LIN {X 0,Y 306.551,Z 155.301,A -85,B 0,C 180,E1 -15794.918,E2 -15794.918} C_VEL
LIN {X 0,Y 305.506,Z 155.43,A -85,B 0,C 180,E1 -15796.018,E2 -15796.018} C_VEL
LIN {X 0,Y 305.419,Z 155.438,A -85,B 0,C 180,E1 -15796.391,E2 -15796.391} C_VEL
LIN {X 0,Y 305.452,Z 155.438,A -85,B 0,C 180,E1 -15799.891,E2 -15799.891} C_VEL
LIN {X 0,Y 305.474,Z 155.435,A -85,B 0,C 180,E1 -15803.63,E2 -15803.63} C_VEL
LIN {X 0,Y 305.457,Z 155.432,A -85,B 0,C 180,E1 -15806.482,E2 -15806.482} C_VEL
LIN {X 0,Y 305.455,Z 155.439,A -85,B 0,C 180,E1 -15809.59,E2 -15809.59} C_VEL
LIN {X 0,Y 305.482,Z 155.427,A -85,B 0,C 180,E1 -15812.604,E2 -15812.604} C_VEL
LIN {X 0,Y 305.483,Z 155.435,A -85,B 0,C 180,E1 -15815.536,E2 -15815.536} C_VEL
LIN {X 0,Y 305.475,Z 155.433,A -85,B 0,C 180,E1 -15819.812,E2 -15819.812} C_VEL
LIN {X 0,Y 305.54,Z 155.42,A -85,B 0,C 180,E1 -15823.977,E2 -15823.977} C_VEL
LIN {X 0,Y 305.576,Z 155.419,A -85,B 0,C 180,E1 -15826.703,E2 -15826.703} C_VEL
LIN {X 0,Y 305.742,Z 155.395,A -85,B 0,C 180,E1 -15831.261,E2 -15831.261} C_VEL
LIN {X 0,Y 305.773,Z 155.383,A -85,B 0,C 180,E1 -15833.401,E2 -15833.401} C_VEL
LIN {X 0,Y 305.923,Z 155.375,A -85,B 0,C 180,E1 -15838.683,E2 -15838.683} C_VEL
LIN {X 0,Y 305.923,Z 155.377,A -85,B 0,C 180,E1 -15841.316,E2 -15841.316} C_VEL
LIN {X 0,Y 305.775,Z 155.396,A -85,B 0,C 180,E1 -15846.599,E2 -15846.599} C_VEL
LIN {X 0,Y 305.684,Z 155.408,A -85,B 0,C 180,E1 -15849.261,E2 -15849.261} C_VEL
LIN {X 0,Y 305.576,Z 155.421,A -85,B 0,C 180,E1 -15853.297,E2 -15853.297} C_VEL
LIN {X 0,Y 305.54,Z 155.423,A -85,B 0,C 180,E1 -15856.023,E2 -15856.023} C_VEL
LIN {X 0,Y 305.474,Z 155.433,A -85,B 0,C 180,E1 -15860.188,E2 -15860.188} C_VEL
LIN {X 0,Y 305.482,Z 155.435,A -85,B 0,C 180,E1 -15864.463,E2 -15864.463} C_VEL
LIN {X 0,Y 305.481,Z 155.432,A -85,B 0,C 180,E1 -15867.395,E2 -15867.395} C_VEL
LIN {X 0,Y 305.454,Z 155.44,A -85,B 0,C 180,E1 -15870.41,E2 -15870.41} C_VEL
LIN {X 0,Y 305.456,Z 155.437,A -85,B 0,C 180,E1 -15874.079,E2 -15874.079} C_VEL
LIN {X 0,Y 305.467,Z 155.436,A -85,B 0,C 180,E1 -15876.741,E2 -15876.741} C_VEL
LIN {X 0,Y 305.447,Z 155.438,A -85,B 0,C 180,E1 -15880.601,E2 -15880.601} C_VEL
LIN {X 0,Y 305.419,Z 155.44,A -85,B 0,C 180,E1 -15883.656,E2 -15883.656} C_VEL
LIN {X 0,Y 305.449,Z 155.434,A -85,B 0,C 180,E1 -15887.416,E2 -15887.416} C_VEL
LIN {X 0,Y 305.49,Z 155.431,A -85,B 0,C 180,E1 -15891.602,E2 -15891.602} C_VEL
LIN {X 0,Y 305.458,Z 155.437,A -85,B 0,C 180,E1 -15894.888,E2 -15894.888} C_VEL
LIN {X 0,Y 305.514,Z 155.509,A -85,B 0,C 180,E1 -15897.229,E2 -15897.229} C_VEL
LIN {X 0,Y 308.104,Z 167.27,A -85,B 0,C 180,E1 -15900.722,E2 -15900.722} C_VEL
LIN {X 0,Y 309.757,Z 176.68,A -85,B 0,C 180,E1 -15903.38,E2 -15903.38} C_VEL
LIN {X 0,Y 309.124,Z 182.65,A -85,B 0,C 180,E1 -15904.915,E2 -15904.915} C_VEL
LIN {X 0,Y 313.255,Z 210.257,A -85,B 0,C 180,E1 -15905.903,E2 -15905.903} C_VEL
LIN {X 0,Y 315.301,Z 227.992,A -85,B 0,C 180,E1 -15906.476,E2 -15906.476} C_VEL
LIN {X 0,Y 313.856,Z 291.58,A -85,B 0,C 180,E1 -15907.93,E2 -15907.93} C_VEL
LIN {X 0,Y 313.125,Z 304.866,A -85,B 0,C 180,E1 -15908.481,E2 -15908.481} C_VEL
LIN {X 0,Y 312.062,Z 317.037,A -85,B 0,C 180,E1 -15909.226,E2 -15909.226} C_VEL
LIN {X 0,Y 310.871,Z 328.51,A -85,B 0,C 180,E1 -15910.179,E2 -15910.179} C_VEL
LIN {X 0,Y 309.461,Z 340.297,A -85,B 0,C 180,E1 -15911.463,E2 -15911.463} C_VEL
LIN {X 0,Y 308.023,Z 350.876,A -85,B 0,C 180,E1 -15912.918,E2 -15912.918} C_VEL
LIN {X 0,Y 307.034,Z 359.54,A -85,B 0,C 180,E1 -15914.399,E2 -15914.399} C_VEL
LIN {X 0,Y 305.962,Z 367.513,A -85,B 0,C 180,E1 -15916.045,E2 -15916.045} C_VEL
LIN {X 0,Y 304.92,Z 375.297,A -85,B 0,C 180,E1 -15918.029,E2 -15918.029} C_VEL
LIN {X 0,Y 304.28,Z 381.547,A -85,B 0,C 180,E1 -15920.026,E2 -15920.026} C_VEL
LIN {X 0,Y 303.88,Z 386.51,A -85,B 0,C 180,E1 -15922.025,E2 -15922.025} C_VEL
LIN {X 0,Y 303.73,Z 390.71,A -85,B 0,C 180,E1 -15924.256,E2 -15924.256} C_VEL
LIN {X 0,Y 303.707,Z 393.121,A -85,B 0,C 180,E1 -15926.02,E2 -15926.02} C_VEL
LIN {X 0,Y 303.689,Z 394.432,A -85,B 0,C 180,E1 -15927.348,E2 -15927.348} C_VEL
LIN {X 0,Y 303.699,Z 395.344,A -85,B 0,C 180,E1 -15928.675,E2 -15928.675} C_VEL
LIN {X 0,Y 303.761,Z 395.844,A -85,B 0,C 180,E1 -15930.001,E2 -15930.001} C_VEL
LIN {X 0,Y 303.684,Z 395.908,A -85,B 0,C 180,E1 -15931.327,E2 -15931.327} C_VEL
LIN {X 0,Y 303.656,Z 395.586,A -85,B 0,C 180,E1 -15932.654,E2 -15932.654} C_VEL
LIN {X 0,Y 303.651,Z 394.878,A -85,B 0,C 180,E1 -15933.983,E2 -15933.983} C_VEL
LIN {X 0,Y 303.619,Z 393.522,A -85,B 0,C 180,E1 -15935.533,E2 -15935.533} C_VEL
LIN {X 0,Y 303.915,Z 390.231,A -85,B 0,C 180,E1 -15937.977,E2 -15937.977} C_VEL
LIN {X 0,Y 304.375,Z 386.422,A -85,B 0,C 180,E1 -15939.974,E2 -15939.974} C_VEL
LIN {X 0,Y 305.103,Z 381.502,A -85,B 0,C 180,E1 -15941.966,E2 -15941.966} C_VEL
LIN {X 0,Y 306.325,Z 375.332,A -85,B 0,C 180,E1 -15943.941,E2 -15943.941} C_VEL
LIN {X 0,Y 307.732,Z 367.675,A -85,B 0,C 180,E1 -15945.907,E2 -15945.907} C_VEL
LIN {X 0,Y 309.092,Z 359.858,A -85,B 0,C 180,E1 -15947.535,E2 -15947.535} C_VEL
LIN {X 0,Y 310.844,Z 350.334,A -85,B 0,C 180,E1 -15949.138,E2 -15949.138} C_VEL
LIN {X 0,Y 312.706,Z 339.792,A -85,B 0,C 180,E1 -15950.56,E2 -15950.56} C_VEL
LIN {X 0,Y 314.494,Z 328.047,A -85,B 0,C 180,E1 -15951.81,E2 -15951.81} C_VEL
LIN {X 0,Y 316.168,Z 315.476,A -85,B 0,C 180,E1 -15952.807,E2 -15952.807} C_VEL
LIN {X 0,Y 317.508,Z 302.295,A -85,B 0,C 180,E1 -15953.562,E2 -15953.562} C_VEL
LIN {X 0,Y 318.318,Z 289.851,A -85,B 0,C 180,E1 -15954.027,E2 -15954.027} C_VEL
LIN {X 0,Y 319.87,Z 227.886,A -85,B 0,C 180,E1 -15955.437,E2 -15955.437} C_VEL
LIN {X 0,Y 316.156,Z 205.273,A -85,B 0,C 180,E1 -15956.354,E2 -15956.354} C_VEL
LIN {X 0,Y 311.988,Z 184.189,A -85,B 0,C 180,E1 -15957.307,E2 -15957.307} C_VEL
LIN {X 0,Y 311.433,Z 182.073,A -85,B 0,C 180,E1 -15957.456,E2 -15957.456} C_VEL
LIN {X 0,Y 309.514,Z 172.334,A -85,B 0,C 180,E1 -15960.362,E2 -15960.362} C_VEL
LIN {X 0,Y 307.088,Z 161.825,A -85,B 0,C 180,E1 -15963.682,E2 -15963.682} C_VEL
LIN {X 0,Y 305.495,Z 155.433,A -85,B 0,C 180,E1 -15965.818,E2 -15965.818} C_VEL
LIN {X 0,Y 305.469,Z 155.43,A -85,B 0,C 180,E1 -15968.533,E2 -15968.533} C_VEL
LIN {X 0,Y 305.457,Z 155.433,A -85,B 0,C 180,E1 -15972.586,E2 -15972.586} C_VEL
LIN {X 0,Y 305.424,Z 155.44,A -85,B 0,C 180,E1 -15976.345,E2 -15976.345} C_VEL
LIN {X 0,Y 305.412,Z 155.443,A -85,B 0,C 180,E1 -15979.885,E2 -15979.885} C_VEL
LIN {X 0,Y 305.464,Z 155.437,A -85,B 0,C 180,E1 -15983.637,E2 -15983.637} C_VEL
LIN {X 0,Y 305.467,Z 155.436,A -85,B 0,C 180,E1 -15986.483,E2 -15986.483} C_VEL
LIN {X 0,Y 305.432,Z 155.439,A -85,B 0,C 180,E1 -15989.588,E2 -15989.588} C_VEL
LIN {X 0,Y 305.458,Z 155.436,A -85,B 0,C 180,E1 -15992.603,E2 -15992.603} C_VEL
LIN {X 0,Y 305.475,Z 155.432,A -85,B 0,C 180,E1 -15995.536,E2 -15995.536} C_VEL
LIN {X 0,Y 305.461,Z 155.436,A -85,B 0,C 180,E1 -15998.4,E2 -15998.4} C_VEL
LIN {X 0,Y 305.51,Z 155.421,A -85,B 0,C 180,E1 -16001.213,E2 -16001.213} C_VEL
LIN {X 0,Y 305.571,Z 155.41,A -85,B 0,C 180,E1 -16005.345,E2 -16005.345} C_VEL
LIN {X 0,Y 305.623,Z 155.413,A -85,B 0,C 180,E1 -16009.399,E2 -16009.399} C_VEL
LIN {X 0,Y 305.739,Z 155.389,A -85,B 0,C 180,E1 -16012.073,E2 -16012.073} C_VEL
LIN {X 0,Y 305.654,Z 155.41,A -85,B 0,C 180,E1 -16014.723,E2 -16014.723} C_VEL
LIN {X 0,Y 305.932,Z 155.374,A -85,B 0,C 180,E1 -16018.684,E2 -16018.684} C_VEL
LIN {X 0,Y 305.935,Z 155.375,A -85,B 0,C 180,E1 -16021.316,E2 -16021.316} C_VEL
LIN {X 0,Y 305.787,Z 155.392,A -85,B 0,C 180,E1 -16026.599,E2 -16026.599} C_VEL
LIN {X 0,Y 305.696,Z 155.394,A -85,B 0,C 180,E1 -16029.261,E2 -16029.261} C_VEL
LIN {X 0,Y 305.587,Z 155.412,A -85,B 0,C 180,E1 -16033.296,E2 -16033.296} C_VEL
LIN {X 0,Y 305.553,Z 155.423,A -85,B 0,C 180,E1 -16036.022,E2 -16036.022} C_VEL
LIN {X 0,Y 305.486,Z 155.425,A -85,B 0,C 180,E1 -16040.188,E2 -16040.188} C_VEL
LIN {X 0,Y 305.489,Z 155.429,A -85,B 0,C 180,E1 -16043.039,E2 -16043.039} C_VEL
LIN {X 0,Y 305.476,Z 155.432,A -85,B 0,C 180,E1 -16046.198,E2 -16046.198} C_VEL
LIN {X 0,Y 305.465,Z 155.429,A -85,B 0,C 180,E1 -16049.038,E2 -16049.038} C_VEL
LIN {X 0,Y 305.44,Z 155.435,A -85,B 0,C 180,E1 -16051.953,E2 -16051.953} C_VEL
LIN {X 0,Y 305.465,Z 155.433,A -85,B 0,C 180,E1 -16055.113,E2 -16055.113} C_VEL
LIN {X 0,Y 305.453,Z 155.436,A -85,B 0,C 180,E1 -16058.529,E2 -16058.529} C_VEL
LIN {X 0,Y 305.458,Z 155.424,A -85,B 0,C 180,E1 -16062.586,E2 -16062.586} C_VEL
LIN {X 0,Y 305.429,Z 155.442,A -85,B 0,C 180,E1 -16066.345,E2 -16066.345} C_VEL
LIN {X 0,Y 305.462,Z 155.435,A -85,B 0,C 180,E1 -16069.892,E2 -16069.892} C_VEL
LIN {X 0,Y 305.484,Z 155.434,A -85,B 0,C 180,E1 -16073.632,E2 -16073.632} C_VEL
LIN {X 0,Y 305.481,Z 155.444,A -85,B 0,C 180,E1 -16076.12,E2 -16076.12} C_VEL
LIN {X 0,Y 306.181,Z 158.233,A -85,B 0,C 180,E1 -16077.073,E2 -16077.073} C_VEL
LIN {X 0,Y 315.619,Z 178.208,A -85,B 0,C 180,E1 -16078.583,E2 -16078.583} C_VEL
LIN {X 0,Y 320.869,Z 190.79,A -85,B 0,C 180,E1 -16079.412,E2 -16079.412} C_VEL
LIN {X 0,Y 318.922,Z 264.646,A -85,B 0,C 180,E1 -16081.089,E2 -16081.089} C_VEL
LIN {X 0,Y 318.114,Z 278.09,A -85,B 0,C 180,E1 -16081.64,E2 -16081.64} C_VEL
LIN {X 0,Y 316.947,Z 290.836,A -85,B 0,C 180,E1 -16082.42,E2 -16082.42} C_VEL
LIN {X 0,Y 315.814,Z 301.857,A -85,B 0,C 180,E1 -16083.35,E2 -16083.35} C_VEL
LIN {X 0,Y 314.305,Z 312.622,A -85,B 0,C 180,E1 -16084.504,E2 -16084.504} C_VEL
LIN {X 0,Y 312.461,Z 323.31,A -85,B 0,C 180,E1 -16085.94,E2 -16085.94} C_VEL
LIN {X 0,Y 310.788,Z 333.59,A -85,B 0,C 180,E1 -16087.703,E2 -16087.703} C_VEL
LIN {X 0,Y 309.416,Z 341.439,A -85,B 0,C 180,E1 -16089.385,E2 -16089.385} C_VEL
LIN {X 0,Y 307.799,Z 348.931,A -85,B 0,C 180,E1 -16091.356,E2 -16091.356} C_VEL
LIN {X 0,Y 306.52,Z 354.927,A -85,B 0,C 180,E1 -16093.344,E2 -16093.344} C_VEL
LIN {X 0,Y 305.543,Z 359.651,A -85,B 0,C 180,E1 -16095.343,E2 -16095.343} C_VEL
LIN {X 0,Y 304.823,Z 363.251,A -85,B 0,C 180,E1 -16097.347,E2 -16097.347} C_VEL
LIN {X 0,Y 304.261,Z 365.832,A -85,B 0,C 180,E1 -16099.35,E2 -16099.35} C_VEL
LIN {X 0,Y 304.05,Z 367.039,A -85,B 0,C 180,E1 -16100.687,E2 -16100.687} C_VEL
LIN {X 0,Y 303.936,Z 367.823,A -85,B 0,C 180,E1 -16102.024,E2 -16102.024} C_VEL
LIN {X 0,Y 303.915,Z 368.252,A -85,B 0,C 180,E1 -16103.921,E2 -16103.921} C_VEL
LIN {X 0,Y 303.824,Z 367.797,A -85,B 0,C 180,E1 -16106.02,E2 -16106.02} C_VEL
LIN {X 0,Y 303.764,Z 367.012,A -85,B 0,C 180,E1 -16107.347,E2 -16107.347} C_VEL
LIN {X 0,Y 303.999,Z 364.191,A -85,B 0,C 180,E1 -16109.999,E2 -16109.999} C_VEL
LIN {X 0,Y 304.334,Z 360.97,A -85,B 0,C 180,E1 -16111.984,E2 -16111.984} C_VEL
LIN {X 0,Y 304.854,Z 356.695,A -85,B 0,C 180,E1 -16113.965,E2 -16113.965} C_VEL
LIN {X 0,Y 305.747,Z 350.237,A -85,B 0,C 180,E1 -16116.267,E2 -16116.267} C_VEL
LIN {X 0,Y 306.744,Z 343.147,A -85,B 0,C 180,E1 -16118.232,E2 -16118.232} C_VEL
LIN {X 0,Y 307.877,Z 335.937,A -85,B 0,C 180,E1 -16119.857,E2 -16119.857} C_VEL
LIN {X 0,Y 308.713,Z 329.148,A -85,B 0,C 180,E1 -16121.156,E2 -16121.156} C_VEL
LIN {X 0,Y 310.118,Z 318.516,A -85,B 0,C 180,E1 -16122.807,E2 -16122.807} C_VEL
LIN {X 0,Y 311.431,Z 307.191,A -85,B 0,C 180,E1 -16124.205,E2 -16124.205} C_VEL
LIN {X 0,Y 312.562,Z 295.58,A -85,B 0,C 180,E1 -16125.318,E2 -16125.318} C_VEL
LIN {X 0,Y 313.407,Z 283.539,A -85,B 0,C 180,E1 -16126.193,E2 -16126.193} C_VEL
LIN {X 0,Y 314.141,Z 270.385,A -85,B 0,C 180,E1 -16126.865,E2 -16126.865} C_VEL
LIN {X 0,Y 314.557,Z 256.796,A -85,B 0,C 180,E1 -16127.277,E2 -16127.277} C_VEL
LIN {X 0,Y 316.158,Z 186.608,A -85,B 0,C 180,E1 -16128.846,E2 -16128.846} C_VEL
LIN {X 0,Y 314.888,Z 180.875,A -85,B 0,C 180,E1 -16129.078,E2 -16129.078} C_VEL
LIN {X 0,Y 307.233,Z 160.574,A -85,B 0,C 180,E1 -16130.17,E2 -16130.17} C_VEL
LIN {X 0,Y 305.968,Z 157.454,A -85,B 0,C 180,E1 -16130.371,E2 -16130.371} C_VEL
LIN {X 0,Y 305.517,Z 155.429,A -85,B 0,C 180,E1 -16131.063,E2 -16131.063} C_VEL
LIN {X 0,Y 305.504,Z 155.432,A -85,B 0,C 180,E1 -16134.46,E2 -16134.46} C_VEL
LIN {X 0,Y 305.52,Z 155.426,A -85,B 0,C 180,E1 -16137.39,E2 -16137.39} C_VEL
LIN {X 0,Y 305.461,Z 155.436,A -85,B 0,C 180,E1 -16140.407,E2 -16140.407} C_VEL
LIN {X 0,Y 305.461,Z 155.436,A -85,B 0,C 180,E1 -16144.077,E2 -16144.077} C_VEL
LIN {X 0,Y 305.476,Z 155.431,A -85,B 0,C 180,E1 -16146.737,E2 -16146.737} C_VEL
LIN {X 0,Y 305.45,Z 155.434,A -85,B 0,C 180,E1 -16150.598,E2 -16150.598} C_VEL
LIN {X 0,Y 305.42,Z 155.441,A -85,B 0,C 180,E1 -16153.654,E2 -16153.654} C_VEL
LIN {X 0,Y 305.419,Z 155.438,A -85,B 0,C 180,E1 -16156.391,E2 -16156.391} C_VEL
LIN {X 0,Y 304.737,Z 155.524,A -85,B 0,C 180,E1 -16157.491,E2 -16157.491} C_VEL
LIN {X 0,Y 301.866,Z 155.882,A -85,B 0,C 180,E1 -16159.282,E2 -16159.282} C_VEL
LIN {X 0,Y 299.466,Z 156.179,A -85,B 0,C 180,E1 -16160.735,E2 -16160.735} C_VEL
LIN {X 0,Y 298.477,Z 156.305,A -85,B 0,C 180,E1 -16161.86,E2 -16161.86} C_VEL
LIN {X 0,Y 298.418,Z 156.311,A -85,B 0,C 180,E1 -16162.241,E2 -16162.241} C_VEL
LIN {X 0,Y 298.401,Z 156.317,A -85,B 0,C 180,E1 -16165.58,E2 -16165.58} C_VEL
LIN {X 0,Y 298.387,Z 156.314,A -85,B 0,C 180,E1 -16168.79,E2 -16168.79} C_VEL
LIN {X 0,Y 298.439,Z 156.307,A -85,B 0,C 180,E1 -16171.902,E2 -16171.902} C_VEL
LIN {X 0,Y 298.457,Z 156.306,A -85,B 0,C 180,E1 -16174.921,E2 -16174.921} C_VEL
LIN {X 0,Y 298.413,Z 156.311,A -85,B 0,C 180,E1 -16179.312,E2 -16179.312} C_VEL
LIN {X 0,Y 298.456,Z 156.305,A -85,B 0,C 180,E1 -16182.174,E2 -16182.174} C_VEL
LIN {X 0,Y 298.576,Z 156.289,A -85,B 0,C 180,E1 -16184.994,E2 -16184.994} C_VEL
LIN {X 0,Y 298.573,Z 156.295,A -85,B 0,C 180,E1 -16189.146,E2 -16189.146} C_VEL
LIN {X 0,Y 298.686,Z 156.268,A -85,B 0,C 180,E1 -16191.884,E2 -16191.884} C_VEL
LIN {X 0,Y 298.615,Z 156.271,A -85,B 0,C 180,E1 -16194.598,E2 -16194.598} C_VEL
LIN {X 0,Y 298.891,Z 156.251,A -85,B 0,C 180,E1 -16198.652,E2 -16198.652} C_VEL
LIN {X 0,Y 298.891,Z 156.253,A -85,B 0,C 180,E1 -16201.347,E2 -16201.347} C_VEL
LIN {X 0,Y 298.724,Z 156.276,A -85,B 0,C 180,E1 -16206.755,E2 -16206.755} C_VEL
LIN {X 0,Y 298.615,Z 156.287,A -85,B 0,C 180,E1 -16209.482,E2 -16209.482} C_VEL
LIN {X 0,Y 298.535,Z 156.297,A -85,B 0,C 180,E1 -16213.616,E2 -16213.616} C_VEL
LIN {X 0,Y 298.474,Z 156.306,A -85,B 0,C 180,E1 -16216.413,E2 -16216.413} C_VEL
LIN {X 0,Y 298.45,Z 156.307,A -85,B 0,C 180,E1 -16219.627,E2 -16219.627} C_VEL
LIN {X 0,Y 298.416,Z 156.312,A -85,B 0,C 180,E1 -16223.601,E2 -16223.601} C_VEL
LIN {X 0,Y 298.447,Z 156.313,A -85,B 0,C 180,E1 -16226.578,E2 -16226.578} C_VEL
LIN {X 0,Y 298.411,Z 156.313,A -85,B 0,C 180,E1 -16229.642,E2 -16229.642} C_VEL
LIN {X 0,Y 298.387,Z 156.318,A -85,B 0,C 180,E1 -16232.801,E2 -16232.801} C_VEL
LIN {X 0,Y 298.438,Z 156.311,A -85,B 0,C 180,E1 -16236.809,E2 -16236.809} C_VEL
LIN {X 0,Y 298.38,Z 156.316,A -85,B 0,C 180,E1 -16241.089,E2 -16241.089} C_VEL
LIN {X 0,Y 298.392,Z 156.314,A -85,B 0,C 180,E1 -16243.105,E2 -16243.105} C_VEL
LIN {X 0,Y 298.397,Z 156.312,A -85,B 0,C 180,E1 -16246.922,E2 -16246.922} C_VEL
LIN {X 0,Y 298.41,Z 156.312,A -85,B 0,C 180,E1 -16251.005,E2 -16251.005} C_VEL
LIN {X 0,Y 298.427,Z 156.314,A -85,B 0,C 180,E1 -16253.934,E2 -16253.934} C_VEL
LIN {X 0,Y 298.463,Z 156.476,A -85,B 0,C 180,E1 -16256.808,E2 -16256.808} C_VEL
LIN {X 0,Y 300.859,Z 167.223,A -85,B 0,C 180,E1 -16260.1,E2 -16260.1} C_VEL
LIN {X 0,Y 302.772,Z 177.488,A -85,B 0,C 180,E1 -16263.089,E2 -16263.089} C_VEL
LIN {X 0,Y 302.362,Z 182.254,A -85,B 0,C 180,E1 -16264.353,E2 -16264.353} C_VEL
LIN {X 0,Y 306.762,Z 211.709,A -85,B 0,C 180,E1 -16265.456,E2 -16265.456} C_VEL
LIN {X 0,Y 308.696,Z 228.156,A -85,B 0,C 180,E1 -16266.006,E2 -16266.006} C_VEL
LIN {X 0,Y 307.189,Z 291.052,A -85,B 0,C 180,E1 -16267.469,E2 -16267.469} C_VEL
LIN {X 0,Y 306.462,Z 304.412,A -85,B 0,C 180,E1 -16268.034,E2 -16268.034} C_VEL
LIN {X 0,Y 305.297,Z 317.183,A -85,B 0,C 180,E1 -16268.832,E2 -16268.832} C_VEL
LIN {X 0,Y 303.982,Z 329.327,A -85,B 0,C 180,E1 -16269.887,E2 -16269.887} C_VEL
LIN {X 0,Y 302.523,Z 340.894,A -85,B 0,C 180,E1 -16271.197,E2 -16271.197} C_VEL
LIN {X 0,Y 301.042,Z 351.528,A -85,B 0,C 180,E1 -16272.72,E2 -16272.72} C_VEL
LIN {X 0,Y 299.946,Z 360.695,A -85,B 0,C 180,E1 -16274.371,E2 -16274.371} C_VEL
LIN {X 0,Y 298.86,Z 368.395,A -85,B 0,C 180,E1 -16276.054,E2 -16276.054} C_VEL
LIN {X 0,Y 297.799,Z 375.939,A -85,B 0,C 180,E1 -16278.084,E2 -16278.084} C_VEL
LIN {X 0,Y 297.073,Z 382.914,A -85,B 0,C 180,E1 -16280.469,E2 -16280.469} C_VEL
LIN {X 0,Y 296.744,Z 387.511,A -85,B 0,C 180,E1 -16282.517,E2 -16282.517} C_VEL
LIN {X 0,Y 296.62,Z 391.004,A -85,B 0,C 180,E1 -16284.563,E2 -16284.563} C_VEL
LIN {X 0,Y 296.618,Z 392.745,A -85,B 0,C 180,E1 -16285.925,E2 -16285.925} C_VEL
LIN {X 0,Y 296.611,Z 394.068,A -85,B 0,C 180,E1 -16287.285,E2 -16287.285} C_VEL
LIN {X 0,Y 296.611,Z 394.992,A -85,B 0,C 180,E1 -16288.644,E2 -16288.644} C_VEL
LIN {X 0,Y 296.669,Z 395.513,A -85,B 0,C 180,E1 -16290.001,E2 -16290.001} C_VEL
LIN {X 0,Y 296.597,Z 395.591,A -85,B 0,C 180,E1 -16291.359,E2 -16291.359} C_VEL
LIN {X 0,Y 296.578,Z 395.28,A -85,B 0,C 180,E1 -16292.718,E2 -16292.718} C_VEL
LIN {X 0,Y 296.563,Z 394.582,A -85,B 0,C 180,E1 -16294.078,E2 -16294.078} C_VEL
LIN {X 0,Y 296.547,Z 393.419,A -85,B 0,C 180,E1 -16295.51,E2 -16295.51} C_VEL
LIN {X 0,Y 296.857,Z 389.983,A -85,B 0,C 180,E1 -16298.168,E2 -16298.168} C_VEL
LIN {X 0,Y 297.364,Z 386.2,A -85,B 0,C 180,E1 -16300.211,E2 -16300.211} C_VEL
LIN {X 0,Y 298.12,Z 381.308,A -85,B 0,C 180,E1 -16302.251,E2 -16302.251} C_VEL
LIN {X 0,Y 299.426,Z 375.169,A -85,B 0,C 180,E1 -16304.269,E2 -16304.269} C_VEL
LIN {X 0,Y 300.9,Z 367.555,A -85,B 0,C 180,E1 -16306.278,E2 -16306.278} C_VEL
LIN {X 0,Y 302.315,Z 359.785,A -85,B 0,C 180,E1 -16307.941,E2 -16307.941} C_VEL
LIN {X 0,Y 304.14,Z 350.323,A -85,B 0,C 180,E1 -16309.577,E2 -16309.577} C_VEL
LIN {X 0,Y 306.058,Z 339.845,A -85,B 0,C 180,E1 -16311.027,E2 -16311.027} C_VEL
LIN {X 0,Y 307.923,Z 328.207,A -85,B 0,C 180,E1 -16312.3,E2 -16312.3} C_VEL
LIN {X 0,Y 309.664,Z 315.813,A -85,B 0,C 180,E1 -16313.314,E2 -16313.314} C_VEL
LIN {X 0,Y 311.037,Z 302.848,A -85,B 0,C 180,E1 -16314.084,E2 -16314.084} C_VEL
LIN {X 0,Y 311.938,Z 289.634,A -85,B 0,C 180,E1 -16314.6,E2 -16314.6} C_VEL
LIN {X 0,Y 313.568,Z 228.936,A -85,B 0,C 180,E1 -16316.005,E2 -16316.005} C_VEL
LIN {X 0,Y 309.983,Z 206.806,A -85,B 0,C 180,E1 -16316.926,E2 -16316.926} C_VEL
LIN {X 0,Y 305.941,Z 186.404,A -85,B 0,C 180,E1 -16317.881,E2 -16317.881} C_VEL
LIN {X 0,Y 304.258,Z 181.669,A -85,B 0,C 180,E1 -16318.234,E2 -16318.234} C_VEL
LIN {X 0,Y 301.967,Z 170.913,A -85,B 0,C 180,E1 -16321.579,E2 -16321.579} C_VEL
LIN {X 0,Y 299.633,Z 161.081,A -85,B 0,C 180,E1 -16324.821,E2 -16324.821} C_VEL
LIN {X 0,Y 298.442,Z 156.306,A -85,B 0,C 180,E1 -16326.547,E2 -16326.547} C_VEL
LIN {X 0,Y 298.411,Z 156.307,A -85,B 0,C 180,E1 -16329.487,E2 -16329.487} C_VEL
LIN {X 0,Y 298.401,Z 156.314,A -85,B 0,C 180,E1 -16333.104,E2 -16333.104} C_VEL
LIN {X 0,Y 298.373,Z 156.32,A -85,B 0,C 180,E1 -16336.915,E2 -16336.915} C_VEL
LIN {X 0,Y 298.387,Z 156.317,A -85,B 0,C 180,E1 -16341.011,E2 -16341.011} C_VEL
LIN {X 0,Y 298.406,Z 156.315,A -85,B 0,C 180,E1 -16343.928,E2 -16343.928} C_VEL
LIN {X 0,Y 298.395,Z 156.316,A -85,B 0,C 180,E1 -16347.2,E2 -16347.2} C_VEL
LIN {X 0,Y 298.404,Z 156.316,A -85,B 0,C 180,E1 -16350.625,E2 -16350.625} C_VEL
LIN {X 0,Y 298.441,Z 156.311,A -85,B 0,C 180,E1 -16354.92,E2 -16354.92} C_VEL
LIN {X 0,Y 298.4,Z 156.314,A -85,B 0,C 180,E1 -16357.862,E2 -16357.862} C_VEL
LIN {X 0,Y 298.461,Z 156.296,A -85,B 0,C 180,E1 -16360.752,E2 -16360.752} C_VEL
LIN {X 0,Y 298.512,Z 156.291,A -85,B 0,C 180,E1 -16364.991,E2 -16364.991} C_VEL
LIN {X 0,Y 298.581,Z 156.291,A -85,B 0,C 180,E1 -16369.146,E2 -16369.146} C_VEL
LIN {X 0,Y 298.685,Z 156.267,A -85,B 0,C 180,E1 -16371.884,E2 -16371.884} C_VEL
LIN {X 0,Y 298.625,Z 156.286,A -85,B 0,C 180,E1 -16374.598,E2 -16374.598} C_VEL
LIN {X 0,Y 298.9,Z 156.25,A -85,B 0,C 180,E1 -16378.653,E2 -16378.653} C_VEL
LIN {X 0,Y 298.902,Z 156.251,A -85,B 0,C 180,E1 -16381.347,E2 -16381.347} C_VEL
LIN {X 0,Y 298.736,Z 156.271,A -85,B 0,C 180,E1 -16386.755,E2 -16386.755} C_VEL
LIN {X 0,Y 298.628,Z 156.276,A -85,B 0,C 180,E1 -16389.482,E2 -16389.482} C_VEL
LIN {X 0,Y 298.546,Z 156.286,A -85,B 0,C 180,E1 -16393.616,E2 -16393.616} C_VEL
LIN {X 0,Y 298.486,Z 156.303,A -85,B 0,C 180,E1 -16396.412,E2 -16396.412} C_VEL
LIN {X 0,Y 298.448,Z 156.299,A -85,B 0,C 180,E1 -16399.619,E2 -16399.619} C_VEL
LIN {X 0,Y 298.424,Z 156.304,A -85,B 0,C 180,E1 -16403.601,E2 -16403.601} C_VEL
LIN {X 0,Y 298.416,Z 156.313,A -85,B 0,C 180,E1 -16406.582,E2 -16406.582} C_VEL
LIN {X 0,Y 298.403,Z 156.312,A -85,B 0,C 180,E1 -16409.643,E2 -16409.643} C_VEL
LIN {X 0,Y 298.396,Z 156.31,A -85,B 0,C 180,E1 -16412.8,E2 -16412.8} C_VEL
LIN {X 0,Y 298.449,Z 156.304,A -85,B 0,C 180,E1 -16416.807,E2 -16416.807} C_VEL
LIN {X 0,Y 298.39,Z 156.293,A -85,B 0,C 180,E1 -16421.087,E2 -16421.087} C_VEL
LIN {X 0,Y 298.402,Z 156.311,A -85,B 0,C 180,E1 -16423.103,E2 -16423.103} C_VEL
LIN {X 0,Y 298.407,Z 156.313,A -85,B 0,C 180,E1 -16426.921,E2 -16426.921} C_VEL
LIN {X 0,Y 298.403,Z 156.314,A -85,B 0,C 180,E1 -16431.007,E2 -16431.007} C_VEL
LIN {X 0,Y 298.43,Z 156.312,A -85,B 0,C 180,E1 -16434.762,E2 -16434.762} C_VEL
LIN {X 0,Y 298.432,Z 156.424,A -85,B 0,C 180,E1 -16435.512,E2 -16435.512} C_VEL
LIN {X 0,Y 298.956,Z 158.5,A -85,B 0,C 180,E1 -16436.264,E2 -16436.264} C_VEL
LIN {X 0,Y 307.608,Z 176.44,A -85,B 0,C 180,E1 -16437.71,E2 -16437.71} C_VEL
LIN {X 0,Y 314.624,Z 192.703,A -85,B 0,C 180,E1 -16438.853,E2 -16438.853} C_VEL
LIN {X 0,Y 312.552,Z 265.426,A -85,B 0,C 180,E1 -16440.535,E2 -16440.535} C_VEL
LIN {X 0,Y 311.714,Z 278.712,A -85,B 0,C 180,E1 -16441.096,E2 -16441.096} C_VEL
LIN {X 0,Y 310.467,Z 291.692,A -85,B 0,C 180,E1 -16441.912,E2 -16441.912} C_VEL
LIN {X 0,Y 309.148,Z 303.524,A -85,B 0,C 180,E1 -16442.955,E2 -16442.955} C_VEL
LIN {X 0,Y 307.47,Z 315.017,A -85,B 0,C 180,E1 -16444.259,E2 -16444.259} C_VEL
LIN {X 0,Y 305.623,Z 325.341,A -85,B 0,C 180,E1 -16445.728,E2 -16445.728} C_VEL
LIN {X 0,Y 304.126,Z 333.756,A -85,B 0,C 180,E1 -16447.227,E2 -16447.227} C_VEL
LIN {X 0,Y 302.426,Z 342.844,A -85,B 0,C 180,E1 -16449.243,E2 -16449.243} C_VEL
LIN {X 0,Y 300.775,Z 350.144,A -85,B 0,C 180,E1 -16451.258,E2 -16451.258} C_VEL
LIN {X 0,Y 299.643,Z 355.069,A -85,B 0,C 180,E1 -16452.95,E2 -16452.95} C_VEL
LIN {X 0,Y 298.59,Z 359.832,A -85,B 0,C 180,E1 -16454.994,E2 -16454.994} C_VEL
LIN {X 0,Y 297.829,Z 363.468,A -85,B 0,C 180,E1 -16457.045,E2 -16457.045} C_VEL
LIN {X 0,Y 297.241,Z 366.083,A -85,B 0,C 180,E1 -16459.096,E2 -16459.096} C_VEL
LIN {X 0,Y 296.989,Z 367.308,A -85,B 0,C 180,E1 -16460.464,E2 -16460.464} C_VEL
LIN {X 0,Y 296.855,Z 368.123,A -85,B 0,C 180,E1 -16461.832,E2 -16461.832} C_VEL
LIN {X 0,Y 296.827,Z 368.582,A -85,B 0,C 180,E1 -16463.959,E2 -16463.959} C_VEL
LIN {X 0,Y 296.734,Z 368.145,A -85,B 0,C 180,E1 -16465.924,E2 -16465.924} C_VEL
LIN {X 0,Y 296.686,Z 367.389,A -85,B 0,C 180,E1 -16467.283,E2 -16467.283} C_VEL
LIN {X 0,Y 296.904,Z 364.606,A -85,B 0,C 180,E1 -16469.999,E2 -16469.999} C_VEL
LIN {X 0,Y 297.273,Z 361.417,A -85,B 0,C 180,E1 -16472.031,E2 -16472.031} C_VEL
LIN {X 0,Y 297.814,Z 357.18,A -85,B 0,C 180,E1 -16474.058,E2 -16474.058} C_VEL
LIN {X 0,Y 298.733,Z 350.771,A -85,B 0,C 180,E1 -16476.415,E2 -16476.415} C_VEL
LIN {X 0,Y 299.738,Z 343.744,A -85,B 0,C 180,E1 -16478.425,E2 -16478.425} C_VEL
LIN {X 0,Y 300.927,Z 336.587,A -85,B 0,C 180,E1 -16480.087,E2 -16480.087} C_VEL
LIN {X 0,Y 301.792,Z 329.835,A -85,B 0,C 180,E1 -16481.415,E2 -16481.415} C_VEL
LIN {X 0,Y 303.221,Z 319.589,A -85,B 0,C 180,E1 -16483.063,E2 -16483.063} C_VEL
LIN {X 0,Y 304.592,Z 308.088,A -85,B 0,C 180,E1 -16484.531,E2 -16484.531} C_VEL
LIN {X 0,Y 305.782,Z 296.689,A -85,B 0,C 180,E1 -16485.666,E2 -16485.666} C_VEL
LIN {X 0,Y 306.674,Z 284.904,A -85,B 0,C 180,E1 -16486.559,E2 -16486.559} C_VEL
LIN {X 0,Y 307.435,Z 272.175,A -85,B 0,C 180,E1 -16487.244,E2 -16487.244} C_VEL
LIN {X 0,Y 307.886,Z 259.443,A -85,B 0,C 180,E1 -16487.675,E2 -16487.675} C_VEL
LIN {X 0,Y 309.545,Z 187.374,A -85,B 0,C 180,E1 -16489.324,E2 -16489.324} C_VEL
LIN {X 0,Y 308.414,Z 182.75,A -85,B 0,C 180,E1 -16489.525,E2 -16489.525} C_VEL
LIN {X 0,Y 301.23,Z 163.738,A -85,B 0,C 180,E1 -16490.583,E2 -16490.583} C_VEL
LIN {X 0,Y 298.76,Z 157.762,A -85,B 0,C 180,E1 -16490.977,E2 -16490.977} C_VEL
LIN {X 0,Y 298.441,Z 156.311,A -85,B 0,C 180,E1 -16491.498,E2 -16491.498} C_VEL
LIN {X 0,Y 298.483,Z 156.304,A -85,B 0,C 180,E1 -16495.074,E2 -16495.074} C_VEL
LIN {X 0,Y 298.462,Z 156.309,A -85,B 0,C 180,E1 -16498.094,E2 -16498.094} C_VEL
LIN {X 0,Y 298.393,Z 156.317,A -85,B 0,C 180,E1 -16502.015,E2 -16502.015} C_VEL
LIN {X 0,Y 298.428,Z 156.312,A -85,B 0,C 180,E1 -16506.066,E2 -16506.066} C_VEL
LIN {X 0,Y 298.404,Z 156.312,A -85,B 0,C 180,E1 -16509.485,E2 -16509.485} C_VEL
LIN {X 0,Y 298.394,Z 156.313,A -85,B 0,C 180,E1 -16513.102,E2 -16513.102} C_VEL
LIN {X 0,Y 298.397,Z 156.312,A -85,B 0,C 180,E1 -16516.919,E2 -16516.919} C_VEL
LIN {X 0,Y 298.408,Z 156.311,A -85,B 0,C 180,E1 -16521.002,E2 -16521.002} C_VEL
LIN {X 0,Y 298.418,Z 156.311,A -85,B 0,C 180,E1 -16522.241,E2 -16522.241} C_VEL
LIN {X 0,Y 297.812,Z 156.393,A -85,B 0,C 180,E1 -16523.368,E2 -16523.368} C_VEL
LIN {X 0,Y 294.991,Z 156.748,A -85,B 0,C 180,E1 -16525.202,E2 -16525.202} C_VEL
LIN {X 0,Y 292.538,Z 157.05,A -85,B 0,C 180,E1 -16526.69,E2 -16526.69} C_VEL
LIN {X 0,Y 291.448,Z 157.181,A -85,B 0,C 180,E1 -16527.843,E2 -16527.843} C_VEL
LIN {X 0,Y 291.341,Z 157.193,A -85,B 0,C 180,E1 -16528.234,E2 -16528.234} C_VEL
LIN {X 0,Y 291.367,Z 157.191,A -85,B 0,C 180,E1 -16531.156,E2 -16531.156} C_VEL
LIN {X 0,Y 291.392,Z 157.186,A -85,B 0,C 180,E1 -16534.269,E2 -16534.269} C_VEL
LIN {X 0,Y 291.362,Z 157.192,A -85,B 0,C 180,E1 -16537.298,E2 -16537.298} C_VEL
LIN {X 0,Y 291.397,Z 157.185,A -85,B 0,C 180,E1 -16540.266,E2 -16540.266} C_VEL
LIN {X 0,Y 291.488,Z 157.17,A -85,B 0,C 180,E1 -16544.665,E2 -16544.665} C_VEL
LIN {X 0,Y 291.519,Z 157.171,A -85,B 0,C 180,E1 -16548.88,E2 -16548.88} C_VEL
LIN {X 0,Y 291.64,Z 157.146,A -85,B 0,C 180,E1 -16551.686,E2 -16551.686} C_VEL
LIN {X 0,Y 291.585,Z 157.144,A -85,B 0,C 180,E1 -16554.467,E2 -16554.467} C_VEL
LIN {X 0,Y 291.859,Z 157.127,A -85,B 0,C 180,E1 -16558.62,E2 -16558.62} C_VEL
LIN {X 0,Y 291.859,Z 157.128,A -85,B 0,C 180,E1 -16561.38,E2 -16561.38} C_VEL
LIN {X 0,Y 291.676,Z 157.153,A -85,B 0,C 180,E1 -16566.919,E2 -16566.919} C_VEL
LIN {X 0,Y 291.558,Z 157.166,A -85,B 0,C 180,E1 -16569.714,E2 -16569.714} C_VEL
LIN {X 0,Y 291.505,Z 157.173,A -85,B 0,C 180,E1 -16573.951,E2 -16573.951} C_VEL
LIN {X 0,Y 291.418,Z 157.186,A -85,B 0,C 180,E1 -16576.822,E2 -16576.822} C_VEL
LIN {X 0,Y 291.414,Z 157.184,A -85,B 0,C 180,E1 -16579.861,E2 -16579.861} C_VEL
LIN {X 0,Y 291.364,Z 157.193,A -85,B 0,C 180,E1 -16584.208,E2 -16584.208} C_VEL
LIN {X 0,Y 291.395,Z 157.187,A -85,B 0,C 180,E1 -16587.274,E2 -16587.274} C_VEL
LIN {X 0,Y 291.328,Z 157.2,A -85,B 0,C 180,E1 -16590.438,E2 -16590.438} C_VEL
LIN {X 0,Y 291.337,Z 157.195,A -85,B 0,C 180,E1 -16593.699,E2 -16593.699} C_VEL
LIN {X 0,Y 291.368,Z 157.19,A -85,B 0,C 180,E1 -16597.255,E2 -16597.255} C_VEL
LIN {X 0,Y 291.325,Z 157.197,A -85,B 0,C 180,E1 -16600.644,E2 -16600.644} C_VEL
LIN {X 0,Y 291.284,Z 157.203,A -85,B 0,C 180,E1 -16604.403,E2 -16604.403} C_VEL
LIN {X 0,Y 291.321,Z 157.193,A -85,B 0,C 180,E1 -16608.406,E2 -16608.406} C_VEL
LIN {X 0,Y 291.359,Z 157.19,A -85,B 0,C 180,E1 -16611.162,E2 -16611.162} C_VEL
LIN {X 0,Y 291.381,Z 157.192,A -85,B 0,C 180,E1 -16614.631,E2 -16614.631} C_VEL
LIN {X 0,Y 291.419,Z 157.262,A -85,B 0,C 180,E1 -16616.313,E2 -16616.313} C_VEL
LIN {X 0,Y 294.205,Z 169.928,A -85,B 0,C 180,E1 -16620.287,E2 -16620.287} C_VEL
LIN {X 0,Y 295.756,Z 178.303,A -85,B 0,C 180,E1 -16622.783,E2 -16622.783} C_VEL
LIN {X 0,Y 295.597,Z 181.994,A -85,B 0,C 180,E1 -16623.799,E2 -16623.799} C_VEL
LIN {X 0,Y 299.845,Z 210.023,A -85,B 0,C 180,E1 -16624.875,E2 -16624.875} C_VEL
LIN {X 0,Y 302.098,Z 229.047,A -85,B 0,C 180,E1 -16625.532,E2 -16625.532} C_VEL
LIN {X 0,Y 300.525,Z 291.675,A -85,B 0,C 180,E1 -16627.032,E2 -16627.032} C_VEL
LIN {X 0,Y 299.689,Z 305.484,A -85,B 0,C 180,E1 -16627.647,E2 -16627.647} C_VEL
LIN {X 0,Y 298.447,Z 318.352,A -85,B 0,C 180,E1 -16628.503,E2 -16628.503} C_VEL
LIN {X 0,Y 297.097,Z 330.128,A -85,B 0,C 180,E1 -16629.58,E2 -16629.58} C_VEL
LIN {X 0,Y 295.596,Z 341.49,A -85,B 0,C 180,E1 -16630.92,E2 -16630.92} C_VEL
LIN {X 0,Y 294.113,Z 351.72,A -85,B 0,C 180,E1 -16632.443,E2 -16632.443} C_VEL
LIN {X 0,Y 293.011,Z 360.518,A -85,B 0,C 180,E1 -16634.075,E2 -16634.075} C_VEL
LIN {X 0,Y 291.733,Z 369.239,A -85,B 0,C 180,E1 -16636.062,E2 -16636.062} C_VEL
LIN {X 0,Y 290.662,Z 376.578,A -85,B 0,C 180,E1 -16638.141,E2 -16638.141} C_VEL
LIN {X 0,Y 290.04,Z 382.462,A -85,B 0,C 180,E1 -16640.236,E2 -16640.236} C_VEL
LIN {X 0,Y 289.677,Z 387.09,A -85,B 0,C 180,E1 -16642.333,E2 -16642.333} C_VEL
LIN {X 0,Y 289.556,Z 390.608,A -85,B 0,C 180,E1 -16644.43,E2 -16644.43} C_VEL
LIN {X 0,Y 289.534,Z 392.368,A -85,B 0,C 180,E1 -16645.825,E2 -16645.825} C_VEL
LIN {X 0,Y 289.536,Z 393.704,A -85,B 0,C 180,E1 -16647.219,E2 -16647.219} C_VEL
LIN {X 0,Y 289.527,Z 394.639,A -85,B 0,C 180,E1 -16648.61,E2 -16648.61} C_VEL
LIN {X 0,Y 289.579,Z 395.178,A -85,B 0,C 180,E1 -16650.001,E2 -16650.001} C_VEL
LIN {X 0,Y 289.512,Z 395.273,A -85,B 0,C 180,E1 -16651.392,E2 -16651.392} C_VEL
LIN {X 0,Y 289.503,Z 394.974,A -85,B 0,C 180,E1 -16652.784,E2 -16652.784} C_VEL
LIN {X 0,Y 289.434,Z 393.352,A -85,B 0,C 180,E1 -16655.402,E2 -16655.402} C_VEL
LIN {X 0,Y 289.574,Z 391.684,A -85,B 0,C 180,E1 -16656.971,E2 -16656.971} C_VEL
LIN {X 0,Y 289.937,Z 388.617,A -85,B 0,C 180,E1 -16659.066,E2 -16659.066} C_VEL
LIN {X 0,Y 290.607,Z 384.507,A -85,B 0,C 180,E1 -16661.157,E2 -16661.157} C_VEL
LIN {X 0,Y 291.818,Z 378.229,A -85,B 0,C 180,E1 -16663.582,E2 -16663.582} C_VEL
LIN {X 0,Y 293.235,Z 371.418,A -85,B 0,C 180,E1 -16665.643,E2 -16665.643} C_VEL
LIN {X 0,Y 294.781,Z 363.525,A -85,B 0,C 180,E1 -16667.571,E2 -16667.571} C_VEL
LIN {X 0,Y 296.651,Z 354.289,A -85,B 0,C 180,E1 -16669.372,E2 -16669.372} C_VEL
LIN {X 0,Y 298.757,Z 343.625,A -85,B 0,C 180,E1 -16671.024,E2 -16671.024} C_VEL
LIN {X 0,Y 300.67,Z 333.04,A -85,B 0,C 180,E1 -16672.324,E2 -16672.324} C_VEL
LIN {X 0,Y 302.479,Z 321.254,A -85,B 0,C 180,E1 -16673.448,E2 -16673.448} C_VEL
LIN {X 0,Y 304.018,Z 309.013,A -85,B 0,C 180,E1 -16674.317,E2 -16674.317} C_VEL
LIN {X 0,Y 305.234,Z 295.992,A -85,B 0,C 180,E1 -16674.965,E2 -16674.965} C_VEL
LIN {X 0,Y 305.868,Z 281.809,A -85,B 0,C 180,E1 -16675.391,E2 -16675.391} C_VEL
LIN {X 0,Y 307.286,Z 230.011,A -85,B 0,C 180,E1 -16676.596,E2 -16676.596} C_VEL
LIN {X 0,Y 303.916,Z 208.715,A -85,B 0,C 180,E1 -16677.504,E2 -16677.504} C_VEL
LIN {X 0,Y 300.006,Z 188.781,A -85,B 0,C 180,E1 -16678.464,E2 -16678.464} C_VEL
LIN {X 0,Y 297.032,Z 181.328,A -85,B 0,C 180,E1 -16679.041,E2 -16679.041} C_VEL
LIN {X 0,Y 294.385,Z 169.222,A -85,B 0,C 180,E1 -16682.961,E2 -16682.961} C_VEL
LIN {X 0,Y 291.803,Z 158.775,A -85,B 0,C 180,E1 -16686.591,E2 -16686.591} C_VEL
LIN {X 0,Y 291.386,Z 157.185,A -85,B 0,C 180,E1 -16687.256,E2 -16687.256} C_VEL
LIN {X 0,Y 291.336,Z 157.193,A -85,B 0,C 180,E1 -16690.643,E2 -16690.643} C_VEL
LIN {X 0,Y 291.293,Z 157.2,A -85,B 0,C 180,E1 -16694.402,E2 -16694.402} C_VEL
LIN {X 0,Y 291.297,Z 157.2,A -85,B 0,C 180,E1 -16698.412,E2 -16698.412} C_VEL
LIN {X 0,Y 291.336,Z 157.195,A -85,B 0,C 180,E1 -16701.156,E2 -16701.156} C_VEL
LIN {X 0,Y 291.357,Z 157.194,A -85,B 0,C 180,E1 -16704.625,E2 -16704.625} C_VEL
LIN {X 0,Y 291.368,Z 157.191,A -85,B 0,C 180,E1 -16707.95,E2 -16707.95} C_VEL
LIN {X 0,Y 291.346,Z 157.193,A -85,B 0,C 180,E1 -16711.154,E2 -16711.154} C_VEL
LIN {X 0,Y 291.36,Z 157.19,A -85,B 0,C 180,E1 -16714.267,E2 -16714.267} C_VEL
LIN {X 0,Y 291.364,Z 157.191,A -85,B 0,C 180,E1 -16717.298,E2 -16717.298} C_VEL
LIN {X 0,Y 291.39,Z 157.176,A -85,B 0,C 180,E1 -16720.265,E2 -16720.265} C_VEL
LIN {X 0,Y 291.453,Z 157.171,A -85,B 0,C 180,E1 -16724.699,E2 -16724.699} C_VEL
LIN {X 0,Y 291.526,Z 157.17,A -85,B 0,C 180,E1 -16728.88,E2 -16728.88} C_VEL
LIN {X 0,Y 291.631,Z 157.144,A -85,B 0,C 180,E1 -16731.686,E2 -16731.686} C_VEL
LIN {X 0,Y 291.595,Z 157.163,A -85,B 0,C 180,E1 -16734.468,E2 -16734.468} C_VEL
LIN {X 0,Y 291.867,Z 157.125,A -85,B 0,C 180,E1 -16738.62,E2 -16738.62} C_VEL
LIN {X 0,Y 291.87,Z 157.126,A -85,B 0,C 180,E1 -16741.38,E2 -16741.38} C_VEL
LIN {X 0,Y 291.688,Z 157.149,A -85,B 0,C 180,E1 -16746.919,E2 -16746.919} C_VEL
LIN {X 0,Y 291.57,Z 157.157,A -85,B 0,C 180,E1 -16749.714,E2 -16749.714} C_VEL
LIN {X 0,Y 291.517,Z 157.159,A -85,B 0,C 180,E1 -16753.951,E2 -16753.951} C_VEL
LIN {X 0,Y 291.431,Z 157.183,A -85,B 0,C 180,E1 -16756.821,E2 -16756.821} C_VEL
LIN {X 0,Y 291.394,Z 157.178,A -85,B 0,C 180,E1 -16759.842,E2 -16759.842} C_VEL
LIN {X 0,Y 291.363,Z 157.181,A -85,B 0,C 180,E1 -16764.209,E2 -16764.209} C_VEL
LIN {X 0,Y 291.363,Z 157.19,A -85,B 0,C 180,E1 -16767.278,E2 -16767.278} C_VEL
LIN {X 0,Y 291.325,Z 157.195,A -85,B 0,C 180,E1 -16770.439,E2 -16770.439} C_VEL
LIN {X 0,Y 291.347,Z 157.191,A -85,B 0,C 180,E1 -16773.698,E2 -16773.698} C_VEL
LIN {X 0,Y 291.379,Z 157.187,A -85,B 0,C 180,E1 -16777.254,E2 -16777.254} C_VEL
LIN {X 0,Y 291.336,Z 157.173,A -85,B 0,C 180,E1 -16780.642,E2 -16780.642} C_VEL
LIN {X 0,Y 291.294,Z 157.2,A -85,B 0,C 180,E1 -16784.402,E2 -16784.402} C_VEL
LIN {X 0,Y 291.33,Z 157.198,A -85,B 0,C 180,E1 -16788.404,E2 -16788.404} C_VEL
LIN {X 0,Y 291.352,Z 157.192,A -85,B 0,C 180,E1 -16791.157,E2 -16791.157} C_VEL
LIN {X 0,Y 291.424,Z 157.357,A -85,B 0,C 180,E1 -16794.855,E2 -16794.855} C_VEL
LIN {X 0,Y 291.799,Z 158.873,A -85,B 0,C 180,E1 -16795.418,E2 -16795.418} C_VEL
LIN {X 0,Y 301.487,Z 178.56,A -85,B 0,C 180,E1 -16797.1,E2 -16797.1} C_VEL
LIN {X 0,Y 308.354,Z 194.484,A -85,B 0,C 180,E1 -16798.262,E2 -16798.262} C_VEL
LIN {X 0,Y 306.205,Z 266.203,A -85,B 0,C 180,E1 -16799.957,E2 -16799.957} C_VEL
LIN {X 0,Y 305.339,Z 279.34,A -85,B 0,C 180,E1 -16800.528,E2 -16800.528} C_VEL
LIN {X 0,Y 304.135,Z 291.613,A -85,B 0,C 180,E1 -16801.315,E2 -16801.315} C_VEL
LIN {X 0,Y 302.781,Z 303.21,A -85,B 0,C 180,E1 -16802.339,E2 -16802.339} C_VEL
LIN {X 0,Y 301.023,Z 314.821,A -85,B 0,C 180,E1 -16803.666,E2 -16803.666} C_VEL
LIN {X 0,Y 299.052,Z 325.24,A -85,B 0,C 180,E1 -16805.159,E2 -16805.159} C_VEL
LIN {X 0,Y 297.516,Z 333.737,A -85,B 0,C 180,E1 -16806.691,E2 -16806.691} C_VEL
LIN {X 0,Y 295.726,Z 342.896,A -85,B 0,C 180,E1 -16808.75,E2 -16808.75} C_VEL
LIN {X 0,Y 293.976,Z 350.244,A -85,B 0,C 180,E1 -16810.808,E2 -16810.808} C_VEL
LIN {X 0,Y 292.391,Z 356.958,A -85,B 0,C 180,E1 -16813.235,E2 -16813.235} C_VEL
LIN {X 0,Y 291.356,Z 361.367,A -85,B 0,C 180,E1 -16815.327,E2 -16815.327} C_VEL
LIN {X 0,Y 290.61,Z 364.691,A -85,B 0,C 180,E1 -16817.428,E2 -16817.428} C_VEL
LIN {X 0,Y 289.947,Z 367.576,A -85,B 0,C 180,E1 -16820.23,E2 -16820.23} C_VEL
LIN {X 0,Y 289.796,Z 368.418,A -85,B 0,C 180,E1 -16821.632,E2 -16821.632} C_VEL
LIN {X 0,Y 289.75,Z 368.901,A -85,B 0,C 180,E1 -16823.975,E2 -16823.975} C_VEL
LIN {X 0,Y 289.648,Z 368.494,A -85,B 0,C 180,E1 -16825.824,E2 -16825.824} C_VEL
LIN {X 0,Y 289.61,Z 367.761,A -85,B 0,C 180,E1 -16827.217,E2 -16827.217} C_VEL
LIN {X 0,Y 289.64,Z 366.594,A -85,B 0,C 180,E1 -16828.608,E2 -16828.608} C_VEL
LIN {X 0,Y 289.808,Z 365.019,A -85,B 0,C 180,E1 -16829.999,E2 -16829.999} C_VEL
LIN {X 0,Y 290.214,Z 361.864,A -85,B 0,C 180,E1 -16832.08,E2 -16832.08} C_VEL
LIN {X 0,Y 290.758,Z 357.665,A -85,B 0,C 180,E1 -16834.157,E2 -16834.157} C_VEL
LIN {X 0,Y 291.719,Z 351.298,A -85,B 0,C 180,E1 -16836.57,E2 -16836.57} C_VEL
LIN {X 0,Y 292.737,Z 344.34,A -85,B 0,C 180,E1 -16838.628,E2 -16838.628} C_VEL
LIN {X 0,Y 294.134,Z 335.631,A -85,B 0,C 180,E1 -16840.67,E2 -16840.67} C_VEL
LIN {X 0,Y 295.579,Z 325.742,A -85,B 0,C 180,E1 -16842.531,E2 -16842.531} C_VEL
LIN {X 0,Y 297.046,Z 314.882,A -85,B 0,C 180,E1 -16844.14,E2 -16844.14} C_VEL
LIN {X 0,Y 298.492,Z 302.902,A -85,B 0,C 180,E1 -16845.533,E2 -16845.533} C_VEL
LIN {X 0,Y 299.571,Z 290.793,A -85,B 0,C 180,E1 -16846.612,E2 -16846.612} C_VEL
LIN {X 0,Y 300.484,Z 277.305,A -85,B 0,C 180,E1 -16847.48,E2 -16847.48} C_VEL
LIN {X 0,Y 301.126,Z 264.711,A -85,B 0,C 180,E1 -16848.009,E2 -16848.009} C_VEL
LIN {X 0,Y 302.921,Z 188.03,A -85,B 0,C 180,E1 -16849.827,E2 -16849.827} C_VEL
LIN {X 0,Y 301.197,Z 182.504,A -85,B 0,C 180,E1 -16850.107,E2 -16850.107} C_VEL
LIN {X 0,Y 294.717,Z 165.646,A -85,B 0,C 180,E1 -16851.092,E2 -16851.092} C_VEL
LIN {X 0,Y 291.599,Z 158.068,A -85,B 0,C 180,E1 -16851.61,E2 -16851.61} C_VEL
LIN {X 0,Y 291.393,Z 157.189,A -85,B 0,C 180,E1 -16851.952,E2 -16851.952} C_VEL
LIN {X 0,Y 291.415,Z 157.185,A -85,B 0,C 180,E1 -16855.726,E2 -16855.726} C_VEL
LIN {X 0,Y 291.385,Z 157.188,A -85,B 0,C 180,E1 -16859.738,E2 -16859.738} C_VEL
LIN {X 0,Y 291.342,Z 157.193,A -85,B 0,C 180,E1 -16863.697,E2 -16863.697} C_VEL
LIN {X 0,Y 291.381,Z 157.186,A -85,B 0,C 180,E1 -16867.254,E2 -16867.254} C_VEL
LIN {X 0,Y 291.329,Z 157.193,A -85,B 0,C 180,E1 -16870.641,E2 -16870.641} C_VEL
LIN {X 0,Y 291.285,Z 157.2,A -85,B 0,C 180,E1 -16874.4,E2 -16874.4} C_VEL
LIN {X 0,Y 291.32,Z 157.195,A -85,B 0,C 180,E1 -16878.403,E2 -16878.403} C_VEL
LIN {X 0,Y 291.357,Z 157.19,A -85,B 0,C 180,E1 -16881.159,E2 -16881.159} C_VEL
LIN {X 0,Y 291.354,Z 157.191,A -85,B 0,C 180,E1 -16884.625,E2 -16884.625} C_VEL
LIN {X 0,Y 291.341,Z 157.193,A -85,B 0,C 180,E1 -16888.234,E2 -16888.234} C_VEL
LIN {X 0,Y 290.634,Z 157.283,A -85,B 0,C 180,E1 -16889.388,E2 -16889.388} C_VEL
LIN {X 0,Y 287.797,Z 157.636,A -85,B 0,C 180,E1 -16891.269,E2 -16891.269} C_VEL
LIN {X 0,Y 285.418,Z 157.93,A -85,B 0,C 180,E1 -16892.796,E2 -16892.796} C_VEL
LIN {X 0,Y 284.395,Z 158.059,A -85,B 0,C 180,E1 -16893.978,E2 -16893.978} C_VEL
LIN {X 0,Y 284.308,Z 158.066,A -85,B 0,C 180,E1 -16894.378,E2 -16894.378} C_VEL
LIN {X 0,Y 284.303,Z 158.064,A -85,B 0,C 180,E1 -16898.235,E2 -16898.235} C_VEL
LIN {X 0,Y 284.331,Z 158.069,A -85,B 0,C 180,E1 -16901.256,E2 -16901.256} C_VEL
LIN {X 0,Y 284.453,Z 158.051,A -85,B 0,C 180,E1 -16905.696,E2 -16905.696} C_VEL
LIN {X 0,Y 284.504,Z 158.04,A -85,B 0,C 180,E1 -16910.042,E2 -16910.042} C_VEL
LIN {X 0,Y 284.63,Z 158.015,A -85,B 0,C 180,E1 -16912.908,E2 -16912.908} C_VEL
LIN {X 0,Y 284.826,Z 158.002,A -85,B 0,C 180,E1 -16918.586,E2 -16918.586} C_VEL
LIN {X 0,Y 284.826,Z 158.004,A -85,B 0,C 180,E1 -16921.414,E2 -16921.414} C_VEL
LIN {X 0,Y 284.631,Z 158.03,A -85,B 0,C 180,E1 -16927.092,E2 -16927.092} C_VEL
LIN {X 0,Y 284.504,Z 158.044,A -85,B 0,C 180,E1 -16929.957,E2 -16929.957} C_VEL
LIN {X 0,Y 284.453,Z 158.053,A -85,B 0,C 180,E1 -16934.304,E2 -16934.304} C_VEL
LIN {X 0,Y 284.331,Z 158.071,A -85,B 0,C 180,E1 -16938.743,E2 -16938.743} C_VEL
LIN {X 0,Y 284.303,Z 158.07,A -85,B 0,C 180,E1 -16941.765,E2 -16941.765} C_VEL
LIN {X 0,Y 284.319,Z 158.071,A -85,B 0,C 180,E1 -16944.848,E2 -16944.848} C_VEL
LIN {X 0,Y 284.31,Z 158.071,A -85,B 0,C 180,E1 -16948.013,E2 -16948.013} C_VEL
LIN {X 0,Y 284.287,Z 158.073,A -85,B 0,C 180,E1 -16951.275,E2 -16951.275} C_VEL
LIN {X 0,Y 284.333,Z 158.067,A -85,B 0,C 180,E1 -16955.349,E2 -16955.349} C_VEL
LIN {X 0,Y 284.304,Z 158.074,A -85,B 0,C 180,E1 -16958.17,E2 -16958.17} C_VEL
LIN {X 0,Y 284.263,Z 158.078,A -85,B 0,C 180,E1 -16962.126,E2 -16962.126} C_VEL
LIN {X 0,Y 284.25,Z 158.079,A -85,B 0,C 180,E1 -16966.191,E2 -16966.191} C_VEL
LIN {X 0,Y 284.302,Z 158.073,A -85,B 0,C 180,E1 -16970.025,E2 -16970.025} C_VEL
LIN {X 0,Y 284.34,Z 158.069,A -85,B 0,C 180,E1 -16973.617,E2 -16973.617} C_VEL
LIN {X 0,Y 284.36,Z 158.221,A -85,B 0,C 180,E1 -16975.843,E2 -16975.843} C_VEL
LIN {X 0,Y 286.82,Z 169.074,A -85,B 0,C 180,E1 -16979.37,E2 -16979.37} C_VEL
LIN {X 0,Y 288.736,Z 179.09,A -85,B 0,C 180,E1 -16982.455,E2 -16982.455} C_VEL
LIN {X 0,Y 288.87,Z 181.67,A -85,B 0,C 180,E1 -16983.204,E2 -16983.204} C_VEL
LIN {X 0,Y 292.965,Z 208.226,A -85,B 0,C 180,E1 -16984.264,E2 -16984.264} C_VEL
LIN {X 0,Y 295.509,Z 229.198,A -85,B 0,C 180,E1 -16985.018,E2 -16985.018} C_VEL
LIN {X 0,Y 293.905,Z 291.126,A -85,B 0,C 180,E1 -16986.53,E2 -16986.53} C_VEL
LIN {X 0,Y 293.07,Z 305.016,A -85,B 0,C 180,E1 -16987.16,E2 -16987.16} C_VEL
LIN {X 0,Y 291.823,Z 317.427,A -85,B 0,C 180,E1 -16987.99,E2 -16987.99} C_VEL
LIN {X 0,Y 290.427,Z 329.33,A -85,B 0,C 180,E1 -16989.09,E2 -16989.09} C_VEL
LIN {X 0,Y 288.872,Z 340.779,A -85,B 0,C 180,E1 -16990.458,E2 -16990.458} C_VEL
LIN {X 0,Y 287.256,Z 351.091,A -85,B 0,C 180,E1 -16992.01,E2 -16992.01} C_VEL
LIN {X 0,Y 286.079,Z 360.323,A -85,B 0,C 180,E1 -16993.762,E2 -16993.762} C_VEL
LIN {X 0,Y 284.774,Z 368.71,A -85,B 0,C 180,E1 -16995.714,E2 -16995.714} C_VEL
LIN {X 0,Y 283.68,Z 376.087,A -85,B 0,C 180,E1 -16997.845,E2 -16997.845} C_VEL
LIN {X 0,Y 282.999,Z 382.006,A -85,B 0,C 180,E1 -16999.99,E2 -16999.99} C_VEL
LIN {X 0,Y 282.611,Z 386.665,A -85,B 0,C 180,E1 -17002.14,E2 -17002.14} C_VEL
LIN {X 0,Y 282.463,Z 390.381,A -85,B 0,C 180,E1 -17004.411,E2 -17004.411} C_VEL
LIN {X 0,Y 282.461,Z 393.34,A -85,B 0,C 180,E1 -17007.149,E2 -17007.149} C_VEL
LIN {X 0,Y 282.445,Z 394.287,A -85,B 0,C 180,E1 -17008.576,E2 -17008.576} C_VEL
LIN {X 0,Y 282.492,Z 394.841,A -85,B 0,C 180,E1 -17010.001,E2 -17010.001} C_VEL
LIN {X 0,Y 282.43,Z 394.955,A -85,B 0,C 180,E1 -17011.427,E2 -17011.427} C_VEL
LIN {X 0,Y 282.427,Z 394.668,A -85,B 0,C 180,E1 -17012.854,E2 -17012.854} C_VEL
LIN {X 0,Y 282.385,Z 392.926,A -85,B 0,C 180,E1 -17015.715,E2 -17015.715} C_VEL
LIN {X 0,Y 282.499,Z 391.425,A -85,B 0,C 180,E1 -17017.147,E2 -17017.147} C_VEL
LIN {X 0,Y 282.897,Z 388.383,A -85,B 0,C 180,E1 -17019.294,E2 -17019.294} C_VEL
LIN {X 0,Y 283.586,Z 384.299,A -85,B 0,C 180,E1 -17021.436,E2 -17021.436} C_VEL
LIN {X 0,Y 284.877,Z 378.053,A -85,B 0,C 180,E1 -17023.919,E2 -17023.919} C_VEL
LIN {X 0,Y 286.359,Z 371.276,A -85,B 0,C 180,E1 -17026.029,E2 -17026.029} C_VEL
LIN {X 0,Y 287.916,Z 363.733,A -85,B 0,C 180,E1 -17027.927,E2 -17027.927} C_VEL
LIN {X 0,Y 289.955,Z 354.255,A -85,B 0,C 180,E1 -17029.837,E2 -17029.837} C_VEL
LIN {X 0,Y 292.132,Z 343.65,A -85,B 0,C 180,E1 -17031.524,E2 -17031.524} C_VEL
LIN {X 0,Y 294.13,Z 333.14,A -85,B 0,C 180,E1 -17032.849,E2 -17032.849} C_VEL
LIN {X 0,Y 296.005,Z 321.521,A -85,B 0,C 180,E1 -17033.992,E2 -17033.992} C_VEL
LIN {X 0,Y 297.588,Z 309.462,A -85,B 0,C 180,E1 -17034.878,E2 -17034.878} C_VEL
LIN {X 0,Y 298.925,Z 295.776,A -85,B 0,C 180,E1 -17035.58,E2 -17035.58} C_VEL
LIN {X 0,Y 299.589,Z 281.51,A -85,B 0,C 180,E1 -17036.017,E2 -17036.017} C_VEL
LIN {X 0,Y 300.989,Z 230.443,A -85,B 0,C 180,E1 -17037.234,E2 -17037.234} C_VEL
LIN {X 0,Y 297.704,Z 209.723,A -85,B 0,C 180,E1 -17038.15,E2 -17038.15} C_VEL
LIN {X 0,Y 294.174,Z 191.491,A -85,B 0,C 180,E1 -17039.054,E2 -17039.054} C_VEL
LIN {X 0,Y 289.791,Z 181.006,A -85,B 0,C 180,E1 -17039.893,E2 -17039.893} C_VEL
LIN {X 0,Y 287.267,Z 169.624,A -85,B 0,C 180,E1 -17043.715,E2 -17043.715} C_VEL
LIN {X 0,Y 284.794,Z 159.773,A -85,B 0,C 180,E1 -17047.265,E2 -17047.265} C_VEL
LIN {X 0,Y 284.316,Z 158.069,A -85,B 0,C 180,E1 -17047.956,E2 -17047.956} C_VEL
LIN {X 0,Y 284.274,Z 158.074,A -85,B 0,C 180,E1 -17051.876,E2 -17051.876} C_VEL
LIN {X 0,Y 284.24,Z 158.079,A -85,B 0,C 180,E1 -17056.186,E2 -17056.186} C_VEL
LIN {X 0,Y 284.285,Z 158.074,A -85,B 0,C 180,E1 -17060.03,E2 -17060.03} C_VEL
LIN {X 0,Y 284.323,Z 158.071,A -85,B 0,C 180,E1 -17063.613,E2 -17063.613} C_VEL
LIN {X 0,Y 284.308,Z 158.071,A -85,B 0,C 180,E1 -17067.191,E2 -17067.191} C_VEL
LIN {X 0,Y 284.339,Z 158.067,A -85,B 0,C 180,E1 -17070.374,E2 -17070.374} C_VEL
LIN {X 0,Y 284.307,Z 158.068,A -85,B 0,C 180,E1 -17073.58,E2 -17073.58} C_VEL
LIN {X 0,Y 284.329,Z 158.066,A -85,B 0,C 180,E1 -17076.704,E2 -17076.704} C_VEL
LIN {X 0,Y 284.336,Z 158.056,A -85,B 0,C 180,E1 -17079.928,E2 -17079.928} C_VEL
LIN {X 0,Y 284.422,Z 158.049,A -85,B 0,C 180,E1 -17084.513,E2 -17084.513} C_VEL
LIN {X 0,Y 284.458,Z 158.052,A -85,B 0,C 180,E1 -17088.6,E2 -17088.6} C_VEL
LIN {X 0,Y 284.582,Z 158.022,A -85,B 0,C 180,E1 -17091.479,E2 -17091.479} C_VEL
LIN {X 0,Y 284.565,Z 158.039,A -85,B 0,C 180,E1 -17094.331,E2 -17094.331} C_VEL
LIN {X 0,Y 284.834,Z 158,A -85,B 0,C 180,E1 -17098.586,E2 -17098.586} C_VEL
LIN {X 0,Y 284.837,Z 158.001,A -85,B 0,C 180,E1 -17101.414,E2 -17101.414} C_VEL
LIN {X 0,Y 284.643,Z 158.026,A -85,B 0,C 180,E1 -17107.092,E2 -17107.092} C_VEL
LIN {X 0,Y 284.516,Z 158.038,A -85,B 0,C 180,E1 -17109.957,E2 -17109.957} C_VEL
LIN {X 0,Y 284.465,Z 158.037,A -85,B 0,C 180,E1 -17114.304,E2 -17114.304} C_VEL
LIN {X 0,Y 284.335,Z 158.059,A -85,B 0,C 180,E1 -17118.743,E2 -17118.743} C_VEL
LIN {X 0,Y 284.331,Z 158.061,A -85,B 0,C 180,E1 -17123.296,E2 -17123.296} C_VEL
LIN {X 0,Y 284.337,Z 158.066,A -85,B 0,C 180,E1 -17127.149,E2 -17127.149} C_VEL
LIN {X 0,Y 284.303,Z 158.069,A -85,B 0,C 180,E1 -17130.093,E2 -17130.093} C_VEL
LIN {X 0,Y 284.308,Z 158.064,A -85,B 0,C 180,E1 -17132.945,E2 -17132.945} C_VEL
LIN {X 0,Y 284.336,Z 158.061,A -85,B 0,C 180,E1 -17136.386,E2 -17136.386} C_VEL
LIN {X 0,Y 284.309,Z 158.053,A -85,B 0,C 180,E1 -17139.994,E2 -17139.994} C_VEL
LIN {X 0,Y 284.25,Z 158.079,A -85,B 0,C 180,E1 -17144.19,E2 -17144.19} C_VEL
LIN {X 0,Y 284.275,Z 158.074,A -85,B 0,C 180,E1 -17148.124,E2 -17148.124} C_VEL
LIN {X 0,Y 284.323,Z 158.07,A -85,B 0,C 180,E1 -17152.279,E2 -17152.279} C_VEL
LIN {X 0,Y 284.332,Z 158.162,A -85,B 0,C 180,E1 -17154.1,E2 -17154.1} C_VEL
LIN {X 0,Y 284.634,Z 159.378,A -85,B 0,C 180,E1 -17154.524,E2 -17154.524} C_VEL
LIN {X 0,Y 293.839,Z 177.499,A -85,B 0,C 180,E1 -17156.191,E2 -17156.191} C_VEL
LIN {X 0,Y 300.75,Z 193.169,A -85,B 0,C 180,E1 -17157.413,E2 -17157.413} C_VEL
LIN {X 0,Y 302.138,Z 196.5,A -85,B 0,C 180,E1 -17157.655,E2 -17157.655} C_VEL
LIN {X 0,Y 299.96,Z 265.83,A -85,B 0,C 180,E1 -17159.313,E2 -17159.313} C_VEL
LIN {X 0,Y 299.086,Z 279.203,A -85,B 0,C 180,E1 -17159.897,E2 -17159.897} C_VEL
LIN {X 0,Y 297.823,Z 291.537,A -85,B 0,C 180,E1 -17160.692,E2 -17160.692} C_VEL
LIN {X 0,Y 296.461,Z 302.888,A -85,B 0,C 180,E1 -17161.697,E2 -17161.697} C_VEL
LIN {X 0,Y 294.609,Z 314.624,A -85,B 0,C 180,E1 -17163.047,E2 -17163.047} C_VEL
LIN {X 0,Y 292.538,Z 325.133,A -85,B 0,C 180,E1 -17164.567,E2 -17164.567} C_VEL
LIN {X 0,Y 290.931,Z 333.705,A -85,B 0,C 180,E1 -17166.131,E2 -17166.131} C_VEL
LIN {X 0,Y 289.329,Z 341.588,A -85,B 0,C 180,E1 -17167.885,E2 -17167.885} C_VEL
LIN {X 0,Y 287.455,Z 349.23,A -85,B 0,C 180,E1 -17169.983,E2 -17169.983} C_VEL
LIN {X 0,Y 285.97,Z 355.355,A -85,B 0,C 180,E1 -17172.108,E2 -17172.108} C_VEL
LIN {X 0,Y 284.732,Z 360.281,A -85,B 0,C 180,E1 -17174.289,E2 -17174.289} C_VEL
LIN {X 0,Y 283.876,Z 363.905,A -85,B 0,C 180,E1 -17176.396,E2 -17176.396} C_VEL
LIN {X 0,Y 283.182,Z 366.589,A -85,B 0,C 180,E1 -17178.547,E2 -17178.547} C_VEL
LIN {X 0,Y 282.728,Z 368.708,A -85,B 0,C 180,E1 -17181.421,E2 -17181.421} C_VEL
LIN {X 0,Y 282.649,Z 369.208,A -85,B 0,C 180,E1 -17184.041,E2 -17184.041} C_VEL
LIN {X 0,Y 282.566,Z 368.841,A -85,B 0,C 180,E1 -17185.72,E2 -17185.72} C_VEL
LIN {X 0,Y 282.535,Z 368.127,A -85,B 0,C 180,E1 -17187.147,E2 -17187.147} C_VEL
LIN {X 0,Y 282.552,Z 366.99,A -85,B 0,C 180,E1 -17188.573,E2 -17188.573} C_VEL
LIN {X 0,Y 282.713,Z 365.432,A -85,B 0,C 180,E1 -17189.999,E2 -17189.999} C_VEL
LIN {X 0,Y 283.156,Z 362.31,A -85,B 0,C 180,E1 -17192.132,E2 -17192.132} C_VEL
LIN {X 0,Y 283.706,Z 358.149,A -85,B 0,C 180,E1 -17194.261,E2 -17194.261} C_VEL
LIN {X 0,Y 284.706,Z 351.82,A -85,B 0,C 180,E1 -17196.732,E2 -17196.732} C_VEL
LIN {X 0,Y 285.74,Z 344.928,A -85,B 0,C 180,E1 -17198.841,E2 -17198.841} C_VEL
LIN {X 0,Y 287.201,Z 336.277,A -85,B 0,C 180,E1 -17200.931,E2 -17200.931} C_VEL
LIN {X 0,Y 288.54,Z 327.431,A -85,B 0,C 180,E1 -17202.661,E2 -17202.661} C_VEL
LIN {X 0,Y 289.868,Z 318.345,A -85,B 0,C 180,E1 -17204.11,E2 -17204.11} C_VEL
LIN {X 0,Y 291.33,Z 306.993,A -85,B 0,C 180,E1 -17205.566,E2 -17205.566} C_VEL
LIN {X 0,Y 292.578,Z 294.992,A -85,B 0,C 180,E1 -17206.752,E2 -17206.752} C_VEL
LIN {X 0,Y 293.569,Z 282.462,A -85,B 0,C 180,E1 -17207.681,E2 -17207.681} C_VEL
LIN {X 0,Y 294.265,Z 270.217,A -85,B 0,C 180,E1 -17208.312,E2 -17208.312} C_VEL
LIN {X 0,Y 294.789,Z 254.652,A -85,B 0,C 180,E1 -17208.773,E2 -17208.773} C_VEL
LIN {X 0,Y 296.355,Z 188.793,A -85,B 0,C 180,E1 -17210.347,E2 -17210.347} C_VEL
LIN {X 0,Y 288.936,Z 169.17,A -85,B 0,C 180,E1 -17211.514,E2 -17211.514} C_VEL
LIN {X 0,Y 284.41,Z 158.514,A -85,B 0,C 180,E1 -17212.237,E2 -17212.237} C_VEL
LIN {X 0,Y 284.349,Z 158.067,A -85,B 0,C 180,E1 -17212.525,E2 -17212.525} C_VEL
LIN {X 0,Y 284.396,Z 158.058,A -85,B 0,C 180,E1 -17217.172,E2 -17217.172} C_VEL
LIN {X 0,Y 284.294,Z 158.069,A -85,B 0,C 180,E1 -17221.272,E2 -17221.272} C_VEL
LIN {X 0,Y 284.358,Z 158.061,A -85,B 0,C 180,E1 -17225.352,E2 -17225.352} C_VEL
LIN {X 0,Y 284.316,Z 158.069,A -85,B 0,C 180,E1 -17228.166,E2 -17228.166} C_VEL
LIN {X 0,Y 284.265,Z 158.077,A -85,B 0,C 180,E1 -17232.123,E2 -17232.123} C_VEL
LIN {X 0,Y 284.25,Z 158.076,A -85,B 0,C 180,E1 -17236.188,E2 -17236.188} C_VEL
LIN {X 0,Y 284.301,Z 158.072,A -85,B 0,C 180,E1 -17240.022,E2 -17240.022} C_VEL
LIN {X 0,Y 284.327,Z 158.068,A -85,B 0,C 180,E1 -17243.613,E2 -17243.613} C_VEL
LIN {X 0,Y 284.301,Z 158.068,A -85,B 0,C 180,E1 -17247.188,E2 -17247.188} C_VEL
LIN {X 0,Y 284.349,Z 158.063,A -85,B 0,C 180,E1 -17250.375,E2 -17250.375} C_VEL
LIN {X 0,Y 284.351,Z 158.064,A -85,B 0,C 180,E1 -17253.584,E2 -17253.584} C_VEL
LIN {X 0,Y 284.308,Z 158.066,A -85,B 0,C 180,E1 -17254.378,E2 -17254.378} C_VEL
LIN {X 0,Y 283.629,Z 158.157,A -85,B 0,C 180,E1 -17255.56,E2 -17255.56} C_VEL
LIN {X 0,Y 280.771,Z 158.509,A -85,B 0,C 180,E1 -17257.484,E2 -17257.484} C_VEL
LIN {X 0,Y 278.368,Z 158.807,A -85,B 0,C 180,E1 -17259.048,E2 -17259.048} C_VEL
LIN {X 0,Y 277.361,Z 158.934,A -85,B 0,C 180,E1 -17260.259,E2 -17260.259} C_VEL
LIN {X 0,Y 277.292,Z 158.942,A -85,B 0,C 180,E1 -17260.669,E2 -17260.669} C_VEL
LIN {X 0,Y 277.399,Z 158.928,A -85,B 0,C 180,E1 -17265.324,E2 -17265.324} C_VEL
LIN {X 0,Y 277.445,Z 158.92,A -85,B 0,C 180,E1 -17269.786,E2 -17269.786} C_VEL
LIN {X 0,Y 277.588,Z 158.892,A -85,B 0,C 180,E1 -17272.727,E2 -17272.727} C_VEL
LIN {X 0,Y 277.793,Z 158.878,A -85,B 0,C 180,E1 -17278.55,E2 -17278.55} C_VEL
LIN {X 0,Y 277.793,Z 158.88,A -85,B 0,C 180,E1 -17281.45,E2 -17281.45} C_VEL
LIN {X 0,Y 277.59,Z 158.906,A -85,B 0,C 180,E1 -17287.272,E2 -17287.272} C_VEL
LIN {X 0,Y 277.445,Z 158.925,A -85,B 0,C 180,E1 -17290.213,E2 -17290.213} C_VEL
LIN {X 0,Y 277.399,Z 158.934,A -85,B 0,C 180,E1 -17294.676,E2 -17294.676} C_VEL
LIN {X 0,Y 277.295,Z 158.944,A -85,B 0,C 180,E1 -17299.237,E2 -17299.237} C_VEL
LIN {X 0,Y 277.282,Z 158.946,A -85,B 0,C 180,E1 -17303.925,E2 -17303.925} C_VEL
LIN {X 0,Y 277.303,Z 158.943,A -85,B 0,C 180,E1 -17307.5,E2 -17307.5} C_VEL
LIN {X 0,Y 277.264,Z 158.953,A -85,B 0,C 180,E1 -17310.482,E2 -17310.482} C_VEL
LIN {X 0,Y 277.239,Z 158.952,A -85,B 0,C 180,E1 -17313.897,E2 -17313.897} C_VEL
LIN {X 0,Y 277.26,Z 158.948,A -85,B 0,C 180,E1 -17317.471,E2 -17317.471} C_VEL
LIN {X 0,Y 277.203,Z 158.954,A -85,B 0,C 180,E1 -17321.238,E2 -17321.238} C_VEL
LIN {X 0,Y 277.195,Z 158.955,A -85,B 0,C 180,E1 -17325.228,E2 -17325.228} C_VEL
LIN {X 0,Y 277.217,Z 158.952,A -85,B 0,C 180,E1 -17329.514,E2 -17329.514} C_VEL
LIN {X 0,Y 277.271,Z 158.948,A -85,B 0,C 180,E1 -17332.533,E2 -17332.533} C_VEL
LIN {X 0,Y 277.307,Z 158.994,A -85,B 0,C 180,E1 -17335.291,E2 -17335.291} C_VEL
LIN {X 0,Y 280.026,Z 171.057,A -85,B 0,C 180,E1 -17339.322,E2 -17339.322} C_VEL
LIN {X 0,Y 281.904,Z 181.251,A -85,B 0,C 180,E1 -17342.531,E2 -17342.531} C_VEL
LIN {X 0,Y 283.278,Z 187.889,A -85,B 0,C 180,E1 -17342.863,E2 -17342.863} C_VEL
LIN {X 0,Y 287.519,Z 217.183,A -85,B 0,C 180,E1 -17344.036,E2 -17344.036} C_VEL
LIN {X 0,Y 288.946,Z 230.326,A -85,B 0,C 180,E1 -17344.507,E2 -17344.507} C_VEL
LIN {X 0,Y 287.289,Z 290.572,A -85,B 0,C 180,E1 -17346.004,E2 -17346.004} C_VEL
LIN {X 0,Y 286.528,Z 303.78,A -85,B 0,C 180,E1 -17346.608,E2 -17346.608} C_VEL
LIN {X 0,Y 285.197,Z 316.456,A -85,B 0,C 180,E1 -17347.451,E2 -17347.451} C_VEL
LIN {X 0,Y 283.755,Z 328.529,A -85,B 0,C 180,E1 -17348.574,E2 -17348.574} C_VEL
LIN {X 0,Y 282.14,Z 340.065,A -85,B 0,C 180,E1 -17349.972,E2 -17349.972} C_VEL
LIN {X 0,Y 280.492,Z 350.459,A -85,B 0,C 180,E1 -17351.56,E2 -17351.56} C_VEL
LIN {X 0,Y 279.307,Z 358.864,A -85,B 0,C 180,E1 -17353.158,E2 -17353.158} C_VEL
LIN {X 0,Y 278.019,Z 366.806,A -85,B 0,C 180,E1 -17354.984,E2 -17354.984} C_VEL
LIN {X 0,Y 276.873,Z 374.466,A -85,B 0,C 180,E1 -17357.169,E2 -17357.169} C_VEL
LIN {X 0,Y 275.95,Z 381.544,A -85,B 0,C 180,E1 -17359.732,E2 -17359.732} C_VEL
LIN {X 0,Y 275.532,Z 386.234,A -85,B 0,C 180,E1 -17361.937,E2 -17361.937} C_VEL
LIN {X 0,Y 275.373,Z 390.247,A -85,B 0,C 180,E1 -17364.472,E2 -17364.472} C_VEL
LIN {X 0,Y 275.388,Z 392.975,A -85,B 0,C 180,E1 -17367.076,E2 -17367.076} C_VEL
LIN {X 0,Y 275.365,Z 393.934,A -85,B 0,C 180,E1 -17368.539,E2 -17368.539} C_VEL
LIN {X 0,Y 275.408,Z 394.501,A -85,B 0,C 180,E1 -17370.001,E2 -17370.001} C_VEL
LIN {X 0,Y 275.351,Z 394.638,A -85,B 0,C 180,E1 -17371.464,E2 -17371.464} C_VEL
LIN {X 0,Y 275.33,Z 394.362,A -85,B 0,C 180,E1 -17372.928,E2 -17372.928} C_VEL
LIN {X 0,Y 275.297,Z 392.643,A -85,B 0,C 180,E1 -17375.862,E2 -17375.862} C_VEL
LIN {X 0,Y 275.448,Z 391.167,A -85,B 0,C 180,E1 -17377.331,E2 -17377.331} C_VEL
LIN {X 0,Y 275.875,Z 388.148,A -85,B 0,C 180,E1 -17379.533,E2 -17379.533} C_VEL
LIN {X 0,Y 276.576,Z 384.089,A -85,B 0,C 180,E1 -17381.73,E2 -17381.73} C_VEL
LIN {X 0,Y 277.965,Z 377.878,A -85,B 0,C 180,E1 -17384.273,E2 -17384.273} C_VEL
LIN {X 0,Y 279.518,Z 371.134,A -85,B 0,C 180,E1 -17386.432,E2 -17386.432} C_VEL
LIN {X 0,Y 281.358,Z 362.617,A -85,B 0,C 180,E1 -17388.614,E2 -17388.614} C_VEL
LIN {X 0,Y 283.27,Z 354.221,A -85,B 0,C 180,E1 -17390.326,E2 -17390.326} C_VEL
LIN {X 0,Y 285.533,Z 343.675,A -85,B 0,C 180,E1 -17392.047,E2 -17392.047} C_VEL
LIN {X 0,Y 287.602,Z 333.24,A -85,B 0,C 180,E1 -17393.398,E2 -17393.398} C_VEL
LIN {X 0,Y 289.548,Z 321.774,A -85,B 0,C 180,E1 -17394.562,E2 -17394.562} C_VEL
LIN {X 0,Y 291.318,Z 308.615,A -85,B 0,C 180,E1 -17395.547,E2 -17395.547} C_VEL
LIN {X 0,Y 292.648,Z 295.53,A -85,B 0,C 180,E1 -17396.223,E2 -17396.223} C_VEL
LIN {X 0,Y 293.296,Z 282.877,A -85,B 0,C 180,E1 -17396.63,E2 -17396.63} C_VEL
LIN {X 0,Y 294.799,Z 231.426,A -85,B 0,C 180,E1 -17397.877,E2 -17397.877} C_VEL
LIN {X 0,Y 291.131,Z 208.33,A -85,B 0,C 180,E1 -17398.938,E2 -17398.938} C_VEL
LIN {X 0,Y 288.388,Z 194.306,A -85,B 0,C 180,E1 -17399.664,E2 -17399.664} C_VEL
LIN {X 0,Y 283.762,Z 183.783,A -85,B 0,C 180,E1 -17400.547,E2 -17400.547} C_VEL
LIN {X 0,Y 282.477,Z 180.59,A -85,B 0,C 180,E1 -17400.833,E2 -17400.833} C_VEL
LIN {X 0,Y 280.345,Z 170.961,A -85,B 0,C 180,E1 -17404.18,E2 -17404.18} C_VEL
LIN {X 0,Y 277.965,Z 161.53,A -85,B 0,C 180,E1 -17407.688,E2 -17407.688} C_VEL
LIN {X 0,Y 277.258,Z 158.942,A -85,B 0,C 180,E1 -17408.706,E2 -17408.706} C_VEL
LIN {X 0,Y 277.212,Z 158.954,A -85,B 0,C 180,E1 -17413.199,E2 -17413.199} C_VEL
LIN {X 0,Y 277.195,Z 158.956,A -85,B 0,C 180,E1 -17417.331,E2 -17417.331} C_VEL
LIN {X 0,Y 277.254,Z 158.951,A -85,B 0,C 180,E1 -17421.796,E2 -17421.796} C_VEL
LIN {X 0,Y 277.28,Z 158.947,A -85,B 0,C 180,E1 -17424.341,E2 -17424.341} C_VEL
LIN {X 0,Y 277.242,Z 158.951,A -85,B 0,C 180,E1 -17427.836,E2 -17427.836} C_VEL
LIN {X 0,Y 277.241,Z 158.949,A -85,B 0,C 180,E1 -17431.207,E2 -17431.207} C_VEL
LIN {X 0,Y 277.248,Z 158.948,A -85,B 0,C 180,E1 -17434.473,E2 -17434.473} C_VEL
LIN {X 0,Y 277.26,Z 158.947,A -85,B 0,C 180,E1 -17437.653,E2 -17437.653} C_VEL
LIN {X 0,Y 277.279,Z 158.934,A -85,B 0,C 180,E1 -17440.762,E2 -17440.762} C_VEL
LIN {X 0,Y 277.368,Z 158.922,A -85,B 0,C 180,E1 -17445.322,E2 -17445.322} C_VEL
LIN {X 0,Y 277.453,Z 158.921,A -85,B 0,C 180,E1 -17449.787,E2 -17449.787} C_VEL
LIN {X 0,Y 277.593,Z 158.9,A -85,B 0,C 180,E1 -17452.728,E2 -17452.728} C_VEL
LIN {X 0,Y 277.8,Z 158.875,A -85,B 0,C 180,E1 -17458.55,E2 -17458.55} C_VEL
LIN {X 0,Y 277.804,Z 158.876,A -85,B 0,C 180,E1 -17461.45,E2 -17461.45} C_VEL
LIN {X 0,Y 277.602,Z 158.9,A -85,B 0,C 180,E1 -17467.272,E2 -17467.272} C_VEL
LIN {X 0,Y 277.46,Z 158.921,A -85,B 0,C 180,E1 -17470.213,E2 -17470.213} C_VEL
LIN {X 0,Y 277.412,Z 158.916,A -85,B 0,C 180,E1 -17474.676,E2 -17474.676} C_VEL
LIN {X 0,Y 277.288,Z 158.934,A -85,B 0,C 180,E1 -17479.238,E2 -17479.238} C_VEL
LIN {X 0,Y 277.286,Z 158.935,A -85,B 0,C 180,E1 -17483.925,E2 -17483.925} C_VEL
LIN {X 0,Y 277.278,Z 158.943,A -85,B 0,C 180,E1 -17487.485,E2 -17487.485} C_VEL
LIN {X 0,Y 277.251,Z 158.949,A -85,B 0,C 180,E1 -17490.473,E2 -17490.473} C_VEL
LIN {X 0,Y 277.25,Z 158.947,A -85,B 0,C 180,E1 -17493.896,E2 -17493.896} C_VEL
LIN {X 0,Y 277.271,Z 158.945,A -85,B 0,C 180,E1 -17497.469,E2 -17497.469} C_VEL
LIN {X 0,Y 277.213,Z 158.929,A -85,B 0,C 180,E1 -17501.236,E2 -17501.236} C_VEL
LIN {X 0,Y 277.205,Z 158.951,A -85,B 0,C 180,E1 -17505.226,E2 -17505.226} C_VEL
LIN {X 0,Y 277.226,Z 158.952,A -85,B 0,C 180,E1 -17509.512,E2 -17509.512} C_VEL
LIN {X 0,Y 277.276,Z 158.947,A -85,B 0,C 180,E1 -17513.296,E2 -17513.296} C_VEL
LIN {X 0,Y 277.486,Z 159.888,A -85,B 0,C 180,E1 -17513.575,E2 -17513.575} C_VEL
LIN {X 0,Y 278.88,Z 162.618,A -85,B 0,C 180,E1 -17513.85,E2 -17513.85} C_VEL
LIN {X 0,Y 285.668,Z 175.447,A -85,B 0,C 180,E1 -17515.128,E2 -17515.128} C_VEL
LIN {X 0,Y 293.41,Z 192.188,A -85,B 0,C 180,E1 -17516.552,E2 -17516.552} C_VEL
LIN {X 0,Y 295.957,Z 198.457,A -85,B 0,C 180,E1 -17517.02,E2 -17517.02} C_VEL
LIN {X 0,Y 293.691,Z 266.621,A -85,B 0,C 180,E1 -17518.685,E2 -17518.685} C_VEL
LIN {X 0,Y 292.787,Z 279.838,A -85,B 0,C 180,E1 -17519.28,E2 -17519.28} C_VEL
LIN {X 0,Y 291.353,Z 293.124,A -85,B 0,C 180,E1 -17520.169,E2 -17520.169} C_VEL
LIN {X 0,Y 289.929,Z 304.175,A -85,B 0,C 180,E1 -17521.197,E2 -17521.197} C_VEL
LIN {X 0,Y 288.006,Z 315.726,A -85,B 0,C 180,E1 -17522.574,E2 -17522.574} C_VEL
LIN {X 0,Y 285.881,Z 326.1,A -85,B 0,C 180,E1 -17524.127,E2 -17524.127} C_VEL
LIN {X 0,Y 284.018,Z 335.384,A -85,B 0,C 180,E1 -17525.901,E2 -17525.901} C_VEL
LIN {X 0,Y 282.091,Z 344.357,A -85,B 0,C 180,E1 -17528.054,E2 -17528.054} C_VEL
LIN {X 0,Y 280.179,Z 351.561,A -85,B 0,C 180,E1 -17530.205,E2 -17530.205} C_VEL
LIN {X 0,Y 278.7,Z 357.284,A -85,B 0,C 180,E1 -17532.385,E2 -17532.385} C_VEL
LIN {X 0,Y 277.616,Z 361.395,A -85,B 0,C 180,E1 -17534.371,E2 -17534.371} C_VEL
LIN {X 0,Y 276.665,Z 365.162,A -85,B 0,C 180,E1 -17536.783,E2 -17536.783} C_VEL
LIN {X 0,Y 275.864,Z 368.114,A -85,B 0,C 180,E1 -17539.726,E2 -17539.726} C_VEL
LIN {X 0,Y 275.657,Z 368.994,A -85,B 0,C 180,E1 -17541.2,E2 -17541.2} C_VEL
LIN {X 0,Y 275.586,Z 369.459,A -85,B 0,C 180,E1 -17542.673,E2 -17542.673} C_VEL
LIN {X 0,Y 275.572,Z 369.51,A -85,B 0,C 180,E1 -17544.144,E2 -17544.144} C_VEL
LIN {X 0,Y 275.462,Z 368.49,A -85,B 0,C 180,E1 -17547.074,E2 -17547.074} C_VEL
LIN {X 0,Y 275.467,Z 367.385,A -85,B 0,C 180,E1 -17548.537,E2 -17548.537} C_VEL
LIN {X 0,Y 275.901,Z 363.896,A -85,B 0,C 180,E1 -17551.458,E2 -17551.458} C_VEL
LIN {X 0,Y 276.446,Z 360.125,A -85,B 0,C 180,E1 -17553.643,E2 -17553.643} C_VEL
LIN {X 0,Y 277.184,Z 355.245,A -85,B 0,C 180,E1 -17555.82,E2 -17555.82} C_VEL
LIN {X 0,Y 278.249,Z 349.104,A -85,B 0,C 180,E1 -17557.984,E2 -17557.984} C_VEL
LIN {X 0,Y 279.469,Z 341.459,A -85,B 0,C 180,E1 -17560.137,E2 -17560.137} C_VEL
LIN {X 0,Y 280.745,Z 333.637,A -85,B 0,C 180,E1 -17561.917,E2 -17561.917} C_VEL
LIN {X 0,Y 282.414,Z 323.386,A -85,B 0,C 180,E1 -17563.795,E2 -17563.795} C_VEL
LIN {X 0,Y 283.797,Z 313.493,A -85,B 0,C 180,E1 -17565.254,E2 -17565.254} C_VEL
LIN {X 0,Y 285.13,Z 303.233,A -85,B 0,C 180,E1 -17566.465,E2 -17566.465} C_VEL
LIN {X 0,Y 286.307,Z 290.991,A -85,B 0,C 180,E1 -17567.59,E2 -17567.59} C_VEL
LIN {X 0,Y 287.241,Z 278.105,A -85,B 0,C 180,E1 -17568.452,E2 -17568.452} C_VEL
LIN {X 0,Y 287.904,Z 265.55,A -85,B 0,C 180,E1 -17569.008,E2 -17569.008} C_VEL
LIN {X 0,Y 289.859,Z 190.499,A -85,B 0,C 180,E1 -17570.862,E2 -17570.862} C_VEL
LIN {X 0,Y 283.033,Z 172.33,A -85,B 0,C 180,E1 -17571.977,E2 -17571.977} C_VEL
LIN {X 0,Y 278.224,Z 161.674,A -85,B 0,C 180,E1 -17572.741,E2 -17572.741} C_VEL
LIN {X 0,Y 277.316,Z 158.943,A -85,B 0,C 180,E1 -17572.941,E2 -17572.941} C_VEL
LIN {X 0,Y 277.358,Z 158.935,A -85,B 0,C 180,E1 -17577.134,E2 -17577.134} C_VEL
LIN {X 0,Y 277.27,Z 158.946,A -85,B 0,C 180,E1 -17580.48,E2 -17580.48} C_VEL
LIN {X 0,Y 277.252,Z 158.949,A -85,B 0,C 180,E1 -17583.893,E2 -17583.893} C_VEL
LIN {X 0,Y 277.272,Z 158.944,A -85,B 0,C 180,E1 -17587.466,E2 -17587.466} C_VEL
LIN {X 0,Y 277.205,Z 158.952,A -85,B 0,C 180,E1 -17591.235,E2 -17591.235} C_VEL
LIN {X 0,Y 277.196,Z 158.955,A -85,B 0,C 180,E1 -17595.225,E2 -17595.225} C_VEL
LIN {X 0,Y 277.217,Z 158.954,A -85,B 0,C 180,E1 -17599.511,E2 -17599.511} C_VEL
LIN {X 0,Y 277.265,Z 158.944,A -85,B 0,C 180,E1 -17602.53,E2 -17602.53} C_VEL
LIN {X 0,Y 277.24,Z 158.948,A -85,B 0,C 180,E1 -17606.103,E2 -17606.103} C_VEL
LIN {X 0,Y 277.254,Z 158.951,A -85,B 0,C 180,E1 -17609.537,E2 -17609.537} C_VEL
LIN {X 0,Y 277.333,Z 158.933,A -85,B 0,C 180,E1 -17612.861,E2 -17612.861} C_VEL
LIN {X 0,Y 277.283,Z 158.944,A -85,B 0,C 180,E1 -17616.075,E2 -17616.075} C_VEL
LIN {X 0,Y 277.292,Z 158.942,A -85,B 0,C 180,E1 -17620.669,E2 -17620.669} C_VEL
LIN {X 0,Y 276.661,Z 159.024,A -85,B 0,C 180,E1 -17621.883,E2 -17621.883} C_VEL
LIN {X 0,Y 273.838,Z 159.374,A -85,B 0,C 180,E1 -17623.862,E2 -17623.862} C_VEL
LIN {X 0,Y 271.429,Z 159.673,A -85,B 0,C 180,E1 -17625.47,E2 -17625.47} C_VEL
LIN {X 0,Y 270.402,Z 159.8,A -85,B 0,C 180,E1 -17626.715,E2 -17626.715} C_VEL
LIN {X 0,Y 270.323,Z 159.807,A -85,B 0,C 180,E1 -17627.137,E2 -17627.137} C_VEL
LIN {X 0,Y 270.518,Z 159.78,A -85,B 0,C 180,E1 -17631.032,E2 -17631.032} C_VEL
LIN {X 0,Y 270.497,Z 159.765,A -85,B 0,C 180,E1 -17634.034,E2 -17634.034} C_VEL
LIN {X 0,Y 270.758,Z 159.754,A -85,B 0,C 180,E1 -17638.512,E2 -17638.512} C_VEL
LIN {X 0,Y 270.759,Z 159.756,A -85,B 0,C 180,E1 -17641.487,E2 -17641.487} C_VEL
LIN {X 0,Y 270.552,Z 159.782,A -85,B 0,C 180,E1 -17647.463,E2 -17647.463} C_VEL
LIN {X 0,Y 270.396,Z 159.804,A -85,B 0,C 180,E1 -17650.483,E2 -17650.483} C_VEL
LIN {X 0,Y 270.358,Z 159.808,A -85,B 0,C 180,E1 -17655.067,E2 -17655.067} C_VEL
LIN {X 0,Y 270.242,Z 159.822,A -85,B 0,C 180,E1 -17659.76,E2 -17659.76} C_VEL
LIN {X 0,Y 270.226,Z 159.826,A -85,B 0,C 180,E1 -17664.59,E2 -17664.59} C_VEL
LIN {X 0,Y 270.236,Z 159.824,A -85,B 0,C 180,E1 -17667.913,E2 -17667.913} C_VEL
LIN {X 0,Y 270.176,Z 159.831,A -85,B 0,C 180,E1 -17671.349,E2 -17671.349} C_VEL
LIN {X 0,Y 270.194,Z 159.83,A -85,B 0,C 180,E1 -17674.907,E2 -17674.907} C_VEL
LIN {X 0,Y 270.19,Z 159.831,A -85,B 0,C 180,E1 -17678.712,E2 -17678.712} C_VEL
LIN {X 0,Y 270.159,Z 159.832,A -85,B 0,C 180,E1 -17683.25,E2 -17683.25} C_VEL
LIN {X 0,Y 270.166,Z 159.828,A -85,B 0,C 180,E1 -17687.443,E2 -17687.443} C_VEL
LIN {X 0,Y 270.202,Z 159.826,A -85,B 0,C 180,E1 -17691.376,E2 -17691.376} C_VEL
LIN {X 0,Y 270.265,Z 159.945,A -85,B 0,C 180,E1 -17694.765,E2 -17694.765} C_VEL
LIN {X 0,Y 272.753,Z 170.967,A -85,B 0,C 180,E1 -17698.575,E2 -17698.575} C_VEL
LIN {X 0,Y 274.707,Z 180.949,A -85,B 0,C 180,E1 -17701.834,E2 -17701.834} C_VEL
LIN {X 0,Y 276.489,Z 186.907,A -85,B 0,C 180,E1 -17702.188,E2 -17702.188} C_VEL
LIN {X 0,Y 280.148,Z 211.256,A -85,B 0,C 180,E1 -17703.215,E2 -17703.215} C_VEL
LIN {X 0,Y 282.416,Z 230.4,A -85,B 0,C 180,E1 -17703.944,E2 -17703.944} C_VEL
LIN {X 0,Y 280.727,Z 290.026,A -85,B 0,C 180,E1 -17705.456,E2 -17705.456} C_VEL
LIN {X 0,Y 279.938,Z 303.308,A -85,B 0,C 180,E1 -17706.072,E2 -17706.072} C_VEL
LIN {X 0,Y 278.668,Z 315.461,A -85,B 0,C 180,E1 -17706.893,E2 -17706.893} C_VEL
LIN {X 0,Y 277.121,Z 327.729,A -85,B 0,C 180,E1 -17708.035,E2 -17708.035} C_VEL
LIN {X 0,Y 275.485,Z 339.357,A -85,B 0,C 180,E1 -17709.467,E2 -17709.467} C_VEL
LIN {X 0,Y 273.743,Z 349.816,A -85,B 0,C 180,E1 -17711.089,E2 -17711.089} C_VEL
LIN {X 0,Y 272.341,Z 359.093,A -85,B 0,C 180,E1 -17712.898,E2 -17712.898} C_VEL
LIN {X 0,Y 270.886,Z 367.648,A -85,B 0,C 180,E1 -17714.964,E2 -17714.964} C_VEL
LIN {X 0,Y 269.717,Z 375.1,A -85,B 0,C 180,E1 -17717.205,E2 -17717.205} C_VEL
LIN {X 0,Y 268.92,Z 381.082,A -85,B 0,C 180,E1 -17719.461,E2 -17719.461} C_VEL
LIN {X 0,Y 268.479,Z 385.803,A -85,B 0,C 180,E1 -17721.724,E2 -17721.724} C_VEL
LIN {X 0,Y 268.298,Z 389.398,A -85,B 0,C 180,E1 -17723.987,E2 -17723.987} C_VEL
LIN {X 0,Y 268.25,Z 391.233,A -85,B 0,C 180,E1 -17725.493,E2 -17725.493} C_VEL
LIN {X 0,Y 268.292,Z 392.609,A -85,B 0,C 180,E1 -17726.998,E2 -17726.998} C_VEL
LIN {X 0,Y 268.288,Z 393.581,A -85,B 0,C 180,E1 -17728.5,E2 -17728.5} C_VEL
LIN {X 0,Y 268.325,Z 394.16,A -85,B 0,C 180,E1 -17730.001,E2 -17730.001} C_VEL
LIN {X 0,Y 268.272,Z 394.321,A -85,B 0,C 180,E1 -17731.503,E2 -17731.503} C_VEL
LIN {X 0,Y 268.235,Z 394.055,A -85,B 0,C 180,E1 -17733.005,E2 -17733.005} C_VEL
LIN {X 0,Y 268.221,Z 392.36,A -85,B 0,C 180,E1 -17736.017,E2 -17736.017} C_VEL
LIN {X 0,Y 268.37,Z 390.907,A -85,B 0,C 180,E1 -17737.525,E2 -17737.525} C_VEL
LIN {X 0,Y 268.83,Z 387.908,A -85,B 0,C 180,E1 -17739.785,E2 -17739.785} C_VEL
LIN {X 0,Y 269.579,Z 383.875,A -85,B 0,C 180,E1 -17742.039,E2 -17742.039} C_VEL
LIN {X 0,Y 271.075,Z 377.703,A -85,B 0,C 180,E1 -17744.643,E2 -17744.643} C_VEL
LIN {X 0,Y 272.703,Z 370.992,A -85,B 0,C 180,E1 -17746.855,E2 -17746.855} C_VEL
LIN {X 0,Y 274.534,Z 362.836,A -85,B 0,C 180,E1 -17749.013,E2 -17749.013} C_VEL
LIN {X 0,Y 276.627,Z 354.185,A -85,B 0,C 180,E1 -17750.837,E2 -17750.837} C_VEL
LIN {X 0,Y 278.966,Z 343.703,A -85,B 0,C 180,E1 -17752.595,E2 -17752.595} C_VEL
LIN {X 0,Y 281.386,Z 331.92,A -85,B 0,C 180,E1 -17754.142,E2 -17754.142} C_VEL
LIN {X 0,Y 283.387,Z 320.082,A -85,B 0,C 180,E1 -17755.329,E2 -17755.329} C_VEL
LIN {X 0,Y 285.119,Z 307.78,A -85,B 0,C 180,E1 -17756.242,E2 -17756.242} C_VEL
LIN {X 0,Y 286.425,Z 295.27,A -85,B 0,C 180,E1 -17756.894,E2 -17756.894} C_VEL
LIN {X 0,Y 287.103,Z 282.475,A -85,B 0,C 180,E1 -17757.314,E2 -17757.314} C_VEL
LIN {X 0,Y 288.66,Z 232.623,A -85,B 0,C 180,E1 -17758.541,E2 -17758.541} C_VEL
LIN {X 0,Y 285.682,Z 213.499,A -85,B 0,C 180,E1 -17759.442,E2 -17759.442} C_VEL
LIN {X 0,Y 282.622,Z 197.042,A -85,B 0,C 180,E1 -17760.303,E2 -17760.303} C_VEL
LIN {X 0,Y 276.489,Z 183.316,A -85,B 0,C 180,E1 -17761.523,E2 -17761.523} C_VEL
LIN {X 0,Y 275.206,Z 180.167,A -85,B 0,C 180,E1 -17761.829,E2 -17761.829} C_VEL
LIN {X 0,Y 272.969,Z 170.332,A -85,B 0,C 180,E1 -17765.401,E2 -17765.401} C_VEL
LIN {X 0,Y 270.656,Z 161.556,A -85,B 0,C 180,E1 -17768.831,E2 -17768.831} C_VEL
LIN {X 0,Y 270.187,Z 159.822,A -85,B 0,C 180,E1 -17769.59,E2 -17769.59} C_VEL
LIN {X 0,Y 270.168,Z 159.832,A -85,B 0,C 180,E1 -17773.249,E2 -17773.249} C_VEL
LIN {X 0,Y 270.154,Z 159.833,A -85,B 0,C 180,E1 -17777.438,E2 -17777.438} C_VEL
LIN {X 0,Y 270.21,Z 159.827,A -85,B 0,C 180,E1 -17781.375,E2 -17781.375} C_VEL
LIN {X 0,Y 270.2,Z 159.828,A -85,B 0,C 180,E1 -17785.094,E2 -17785.094} C_VEL
LIN {X 0,Y 270.187,Z 159.829,A -85,B 0,C 180,E1 -17789.137,E2 -17789.137} C_VEL
LIN {X 0,Y 270.225,Z 159.823,A -85,B 0,C 180,E1 -17792.163,E2 -17792.163} C_VEL
LIN {X 0,Y 270.23,Z 159.823,A -85,B 0,C 180,E1 -17795.543,E2 -17795.543} C_VEL
LIN {X 0,Y 270.222,Z 159.812,A -85,B 0,C 180,E1 -17800.238,E2 -17800.238} C_VEL
LIN {X 0,Y 270.339,Z 159.8,A -85,B 0,C 180,E1 -17804.932,E2 -17804.932} C_VEL
LIN {X 0,Y 270.385,Z 159.803,A -85,B 0,C 180,E1 -17809.517,E2 -17809.517} C_VEL
LIN {X 0,Y 270.554,Z 159.774,A -85,B 0,C 180,E1 -17812.537,E2 -17812.537} C_VEL
LIN {X 0,Y 270.764,Z 159.751,A -85,B 0,C 180,E1 -17818.513,E2 -17818.513} C_VEL
LIN {X 0,Y 270.769,Z 159.751,A -85,B 0,C 180,E1 -17821.487,E2 -17821.487} C_VEL
LIN {X 0,Y 270.564,Z 159.774,A -85,B 0,C 180,E1 -17827.463,E2 -17827.463} C_VEL
LIN {X 0,Y 270.412,Z 159.799,A -85,B 0,C 180,E1 -17830.482,E2 -17830.482} C_VEL
LIN {X 0,Y 270.371,Z 159.795,A -85,B 0,C 180,E1 -17835.067,E2 -17835.067} C_VEL
LIN {X 0,Y 270.227,Z 159.813,A -85,B 0,C 180,E1 -17839.761,E2 -17839.761} C_VEL
LIN {X 0,Y 270.228,Z 159.813,A -85,B 0,C 180,E1 -17844.59,E2 -17844.59} C_VEL
LIN {X 0,Y 270.207,Z 159.823,A -85,B 0,C 180,E1 -17847.916,E2 -17847.916} C_VEL
LIN {X 0,Y 270.177,Z 159.829,A -85,B 0,C 180,E1 -17851.349,E2 -17851.349} C_VEL
LIN {X 0,Y 270.205,Z 159.827,A -85,B 0,C 180,E1 -17854.905,E2 -17854.905} C_VEL
LIN {X 0,Y 270.201,Z 159.824,A -85,B 0,C 180,E1 -17858.71,E2 -17858.71} C_VEL
LIN {X 0,Y 270.175,Z 159.816,A -85,B 0,C 180,E1 -17862.558,E2 -17862.558} C_VEL
LIN {X 0,Y 270.169,Z 159.832,A -85,B 0,C 180,E1 -17866.751,E2 -17866.751} C_VEL
LIN {X 0,Y 270.202,Z 159.827,A -85,B 0,C 180,E1 -17871.289,E2 -17871.289} C_VEL
LIN {X 0,Y 270.24,Z 159.949,A -85,B 0,C 180,E1 -17872.525,E2 -17872.525} C_VEL
LIN {X 0,Y 271.253,Z 162.671,A -85,B 0,C 180,E1 -17872.771,E2 -17872.771} C_VEL
LIN {X 0,Y 272.753,Z 164.977,A -85,B 0,C 180,E1 -17873.062,E2 -17873.062} C_VEL
LIN {X 0,Y 278.296,Z 175.079,A -85,B 0,C 180,E1 -17874.149,E2 -17874.149} C_VEL
LIN {X 0,Y 285.802,Z 190.904,A -85,B 0,C 180,E1 -17875.595,E2 -17875.595} C_VEL
LIN {X 0,Y 289.742,Z 200.258,A -85,B 0,C 180,E1 -17876.345,E2 -17876.345} C_VEL
LIN {X 0,Y 287.528,Z 266.269,A -85,B 0,C 180,E1 -17877.986,E2 -17877.986} C_VEL
LIN {X 0,Y 286.591,Z 279.718,A -85,B 0,C 180,E1 -17878.592,E2 -17878.592} C_VEL
LIN {X 0,Y 285.308,Z 291.4,A -85,B 0,C 180,E1 -17879.363,E2 -17879.363} C_VEL
LIN {X 0,Y 283.678,Z 303.871,A -85,B 0,C 180,E1 -17880.501,E2 -17880.501} C_VEL
LIN {X 0,Y 281.669,Z 315.537,A -85,B 0,C 180,E1 -17881.903,E2 -17881.903} C_VEL
LIN {X 0,Y 279.451,Z 326,A -85,B 0,C 180,E1 -17883.486,E2 -17883.486} C_VEL
LIN {X 0,Y 277.49,Z 335.384,A -85,B 0,C 180,E1 -17885.297,E2 -17885.297} C_VEL
LIN {X 0,Y 275.685,Z 343.325,A -85,B 0,C 180,E1 -17887.2,E2 -17887.2} C_VEL
LIN {X 0,Y 273.723,Z 350.549,A -85,B 0,C 180,E1 -17889.326,E2 -17889.326} C_VEL
LIN {X 0,Y 271.879,Z 357.441,A -85,B 0,C 180,E1 -17891.928,E2 -17891.928} C_VEL
LIN {X 0,Y 270.77,Z 361.303,A -85,B 0,C 180,E1 -17893.815,E2 -17893.815} C_VEL
LIN {X 0,Y 269.688,Z 365.393,A -85,B 0,C 180,E1 -17896.434,E2 -17896.434} C_VEL
LIN {X 0,Y 269.162,Z 367.095,A -85,B 0,C 180,E1 -17897.942,E2 -17897.942} C_VEL
LIN {X 0,Y 268.604,Z 369.279,A -85,B 0,C 180,E1 -17900.967,E2 -17900.967} C_VEL
LIN {X 0,Y 268.505,Z 369.775,A -85,B 0,C 180,E1 -17902.479,E2 -17902.479} C_VEL
LIN {X 0,Y 268.5,Z 369.832,A -85,B 0,C 180,E1 -17904.076,E2 -17904.076} C_VEL
LIN {X 0,Y 268.39,Z 368.852,A -85,B 0,C 180,E1 -17906.997,E2 -17906.997} C_VEL
LIN {X 0,Y 268.385,Z 367.778,A -85,B 0,C 180,E1 -17908.498,E2 -17908.498} C_VEL
LIN {X 0,Y 268.525,Z 366.257,A -85,B 0,C 180,E1 -17909.999,E2 -17909.999} C_VEL
LIN {X 0,Y 269.027,Z 363.202,A -85,B 0,C 180,E1 -17912.244,E2 -17912.244} C_VEL
LIN {X 0,Y 269.594,Z 359.115,A -85,B 0,C 180,E1 -17914.484,E2 -17914.484} C_VEL
LIN {X 0,Y 270.68,Z 352.865,A -85,B 0,C 180,E1 -17917.083,E2 -17917.083} C_VEL
LIN {X 0,Y 271.763,Z 346.076,A -85,B 0,C 180,E1 -17919.3,E2 -17919.3} C_VEL
LIN {X 0,Y 273.359,Z 337.568,A -85,B 0,C 180,E1 -17921.492,E2 -17921.492} C_VEL
LIN {X 0,Y 274.803,Z 328.849,A -85,B 0,C 180,E1 -17923.306,E2 -17923.306} C_VEL
LIN {X 0,Y 276.481,Z 318.115,A -85,B 0,C 180,E1 -17925.101,E2 -17925.101} C_VEL
LIN {X 0,Y 277.979,Z 307.322,A -85,B 0,C 180,E1 -17926.523,E2 -17926.523} C_VEL
LIN {X 0,Y 279.337,Z 295.237,A -85,B 0,C 180,E1 -17927.76,E2 -17927.76} C_VEL
LIN {X 0,Y 280.408,Z 282.583,A -85,B 0,C 180,E1 -17928.729,E2 -17928.729} C_VEL
LIN {X 0,Y 281.168,Z 269.947,A -85,B 0,C 180,E1 -17929.387,E2 -17929.387} C_VEL
LIN {X 0,Y 281.781,Z 252.09,A -85,B 0,C 180,E1 -17929.912,E2 -17929.912} C_VEL
LIN {X 0,Y 283.398,Z 192.266,A -85,B 0,C 180,E1 -17931.397,E2 -17931.397} C_VEL
LIN {X 0,Y 277.23,Z 175.751,A -85,B 0,C 180,E1 -17932.444,E2 -17932.444} C_VEL
LIN {X 0,Y 272.566,Z 165.276,A -85,B 0,C 180,E1 -17933.216,E2 -17933.216} C_VEL
LIN {X 0,Y 270.367,Z 160.458,A -85,B 0,C 180,E1 -17933.587,E2 -17933.587} C_VEL
LIN {X 0,Y 270.269,Z 159.82,A -85,B 0,C 180,E1 -17933.618,E2 -17933.618} C_VEL
LIN {X 0,Y 270.27,Z 159.819,A -85,B 0,C 180,E1 -17937.907,E2 -17937.907} C_VEL
LIN {X 0,Y 270.182,Z 159.827,A -85,B 0,C 180,E1 -17941.346,E2 -17941.346} C_VEL
LIN {X 0,Y 270.211,Z 159.823,A -85,B 0,C 180,E1 -17944.902,E2 -17944.902} C_VEL
LIN {X 0,Y 270.194,Z 159.825,A -85,B 0,C 180,E1 -17948.709,E2 -17948.709} C_VEL
LIN {X 0,Y 270.16,Z 159.831,A -85,B 0,C 180,E1 -17953.247,E2 -17953.247} C_VEL
LIN {X 0,Y 270.166,Z 159.829,A -85,B 0,C 180,E1 -17957.44,E2 -17957.44} C_VEL
LIN {X 0,Y 270.201,Z 159.827,A -85,B 0,C 180,E1 -17961.373,E2 -17961.373} C_VEL
LIN {X 0,Y 270.195,Z 159.828,A -85,B 0,C 180,E1 -17965.093,E2 -17965.093} C_VEL
LIN {X 0,Y 270.193,Z 159.827,A -85,B 0,C 180,E1 -17969.129,E2 -17969.129} C_VEL
LIN {X 0,Y 270.253,Z 159.815,A -85,B 0,C 180,E1 -17972.146,E2 -17972.146} C_VEL
LIN {X 0,Y 270.226,Z 159.827,A -85,B 0,C 180,E1 -17975.538,E2 -17975.538} C_VEL
LIN {X 0,Y 270.242,Z 159.82,A -85,B 0,C 180,E1 -17980.24,E2 -17980.24} C_VEL
LIN {X 0,Y 270.358,Z 159.802,A -85,B 0,C 180,E1 -17984.933,E2 -17984.933} C_VEL
LIN {X 0,Y 270.323,Z 159.807,A -85,B 0,C 180,E1 -17987.137,E2 -17987.137} C_VEL
LIN {X 0,Y 269.679,Z 159.891,A -85,B 0,C 180,E1 -17988.382,E2 -17988.382} C_VEL
LIN {X 0,Y 266.889,Z 160.234,A -85,B 0,C 180,E1 -17990.413,E2 -17990.413} C_VEL
LIN {X 0,Y 264.529,Z 160.518,A -85,B 0,C 180,E1 -17992.063,E2 -17992.063} C_VEL
LIN {X 0,Y 263.537,Z 160.632,A -85,B 0,C 180,E1 -17993.341,E2 -17993.341} C_VEL
LIN {X 0,Y 263.467,Z 160.639,A -85,B 0,C 180,E1 -17993.774,E2 -17993.774} C_VEL
LIN {X 0,Y 263.722,Z 160.63,A -85,B 0,C 180,E1 -17998.473,E2 -17998.473} C_VEL
LIN {X 0,Y 263.722,Z 160.632,A -85,B 0,C 180,E1 -18001.527,E2 -18001.527} C_VEL
LIN {X 0,Y 263.516,Z 160.657,A -85,B 0,C 180,E1 -18007.663,E2 -18007.663} C_VEL
LIN {X 0,Y 263.336,Z 160.684,A -85,B 0,C 180,E1 -18010.767,E2 -18010.767} C_VEL
LIN {X 0,Y 263.3,Z 160.686,A -85,B 0,C 180,E1 -18015.481,E2 -18015.481} C_VEL
LIN {X 0,Y 263.226,Z 160.698,A -85,B 0,C 180,E1 -18020.31,E2 -18020.31} C_VEL
LIN {X 0,Y 263.178,Z 160.703,A -85,B 0,C 180,E1 -18025.294,E2 -18025.294} C_VEL
LIN {X 0,Y 263.147,Z 160.708,A -85,B 0,C 180,E1 -18028.733,E2 -18028.733} C_VEL
LIN {X 0,Y 263.125,Z 160.713,A -85,B 0,C 180,E1 -18032.289,E2 -18032.289} C_VEL
LIN {X 0,Y 263.175,Z 160.705,A -85,B 0,C 180,E1 -18036.764,E2 -18036.764} C_VEL
LIN {X 0,Y 263.118,Z 160.71,A -85,B 0,C 180,E1 -18041.595,E2 -18041.595} C_VEL
LIN {X 0,Y 263.117,Z 160.712,A -85,B 0,C 180,E1 -18046.017,E2 -18046.017} C_VEL
LIN {X 0,Y 263.101,Z 160.714,A -85,B 0,C 180,E1 -18050.129,E2 -18050.129} C_VEL
LIN {X 0,Y 263.288,Z 160.841,A -85,B 0,C 180,E1 -18054.2,E2 -18054.2} C_VEL
LIN {X 0,Y 265.987,Z 173.071,A -85,B 0,C 180,E1 -18058.546,E2 -18058.546} C_VEL
LIN {X 0,Y 267.489,Z 180.607,A -85,B 0,C 180,E1 -18061.085,E2 -18061.085} C_VEL
LIN {X 0,Y 270.174,Z 188.389,A -85,B 0,C 180,E1 -18061.596,E2 -18061.596} C_VEL
LIN {X 0,Y 273.994,Z 214.574,A -85,B 0,C 180,E1 -18062.727,E2 -18062.727} C_VEL
LIN {X 0,Y 275.935,Z 231.275,A -85,B 0,C 180,E1 -18063.38,E2 -18063.38} C_VEL
LIN {X 0,Y 274.209,Z 289.455,A -85,B 0,C 180,E1 -18064.883,E2 -18064.883} C_VEL
LIN {X 0,Y 273.387,Z 302.821,A -85,B 0,C 180,E1 -18065.512,E2 -18065.512} C_VEL
LIN {X 0,Y 272.008,Z 315.584,A -85,B 0,C 180,E1 -18066.394,E2 -18066.394} C_VEL
LIN {X 0,Y 270.547,Z 326.925,A -85,B 0,C 180,E1 -18067.472,E2 -18067.472} C_VEL
LIN {X 0,Y 268.821,Z 338.641,A -85,B 0,C 180,E1 -18068.934,E2 -18068.934} C_VEL
LIN {X 0,Y 267.017,Z 349.169,A -85,B 0,C 180,E1 -18070.594,E2 -18070.594} C_VEL
LIN {X 0,Y 265.558,Z 357.931,A -85,B 0,C 180,E1 -18072.315,E2 -18072.315} C_VEL
LIN {X 0,Y 264.272,Z 365.731,A -85,B 0,C 180,E1 -18074.183,E2 -18074.183} C_VEL
LIN {X 0,Y 262.988,Z 373.482,A -85,B 0,C 180,E1 -18076.479,E2 -18076.479} C_VEL
LIN {X 0,Y 262.125,Z 378.784,A -85,B 0,C 180,E1 -18078.401,E2 -18078.401} C_VEL
LIN {X 0,Y 261.548,Z 383.926,A -85,B 0,C 180,E1 -18080.724,E2 -18080.724} C_VEL
LIN {X 0,Y 261.243,Z 387.913,A -85,B 0,C 180,E1 -18083.048,E2 -18083.048} C_VEL
LIN {X 0,Y 261.163,Z 390.853,A -85,B 0,C 180,E1 -18085.371,E2 -18085.371} C_VEL
LIN {X 0,Y 261.2,Z 392.244,A -85,B 0,C 180,E1 -18086.917,E2 -18086.917} C_VEL
LIN {X 0,Y 261.212,Z 393.229,A -85,B 0,C 180,E1 -18088.46,E2 -18088.46} C_VEL
LIN {X 0,Y 261.246,Z 393.819,A -85,B 0,C 180,E1 -18090.001,E2 -18090.001} C_VEL
LIN {X 0,Y 261.195,Z 394.002,A -85,B 0,C 180,E1 -18091.543,E2 -18091.543} C_VEL
LIN {X 0,Y 261.143,Z 393.749,A -85,B 0,C 180,E1 -18093.087,E2 -18093.087} C_VEL
LIN {X 0,Y 261.146,Z 392.076,A -85,B 0,C 180,E1 -18096.181,E2 -18096.181} C_VEL
LIN {X 0,Y 261.312,Z 390.645,A -85,B 0,C 180,E1 -18097.73,E2 -18097.73} C_VEL
LIN {X 0,Y 261.791,Z 387.666,A -85,B 0,C 180,E1 -18100.051,E2 -18100.051} C_VEL
LIN {X 0,Y 262.596,Z 383.658,A -85,B 0,C 180,E1 -18102.364,E2 -18102.364} C_VEL
LIN {X 0,Y 264.198,Z 377.53,A -85,B 0,C 180,E1 -18105.033,E2 -18105.033} C_VEL
LIN {X 0,Y 265.902,Z 370.867,A -85,B 0,C 180,E1 -18107.295,E2 -18107.295} C_VEL
LIN {X 0,Y 267.82,Z 362.737,A -85,B 0,C 180,E1 -18109.508,E2 -18109.508} C_VEL
LIN {X 0,Y 269.99,Z 354.145,A -85,B 0,C 180,E1 -18111.374,E2 -18111.374} C_VEL
LIN {X 0,Y 272.425,Z 343.735,A -85,B 0,C 180,E1 -18113.168,E2 -18113.168} C_VEL
LIN {X 0,Y 274.934,Z 332.029,A -85,B 0,C 180,E1 -18114.746,E2 -18114.746} C_VEL
LIN {X 0,Y 277.008,Z 320.361,A -85,B 0,C 180,E1 -18115.955,E2 -18115.955} C_VEL
LIN {X 0,Y 278.791,Z 308.246,A -85,B 0,C 180,E1 -18116.885,E2 -18116.885} C_VEL
LIN {X 0,Y 280.21,Z 295.056,A -85,B 0,C 180,E1 -18117.596,E2 -18117.596} C_VEL
LIN {X 0,Y 280.938,Z 282.237,A -85,B 0,C 180,E1 -18118.025,E2 -18118.025} C_VEL
LIN {X 0,Y 282.528,Z 233.717,A -85,B 0,C 180,E1 -18119.241,E2 -18119.241} C_VEL
LIN {X 0,Y 279.13,Z 211.549,A -85,B 0,C 180,E1 -18120.321,E2 -18120.321} C_VEL
LIN {X 0,Y 276.811,Z 199.512,A -85,B 0,C 180,E1 -18120.987,E2 -18120.987} C_VEL
LIN {X 0,Y 269.509,Z 183.388,A -85,B 0,C 180,E1 -18122.505,E2 -18122.505} C_VEL
LIN {X 0,Y 267.943,Z 179.866,A -85,B 0,C 180,E1 -18122.85,E2 -18122.85} C_VEL
LIN {X 0,Y 265.706,Z 170.186,A -85,B 0,C 180,E1 -18126.523,E2 -18126.523} C_VEL
LIN {X 0,Y 263.13,Z 160.707,A -85,B 0,C 180,E1 -18130.432,E2 -18130.432} C_VEL
LIN {X 0,Y 263.106,Z 160.71,A -85,B 0,C 180,E1 -18133.989,E2 -18133.989} C_VEL
LIN {X 0,Y 263.111,Z 160.712,A -85,B 0,C 180,E1 -18138.411,E2 -18138.411} C_VEL
LIN {X 0,Y 263.159,Z 160.706,A -85,B 0,C 180,E1 -18142.103,E2 -18142.103} C_VEL
LIN {X 0,Y 263.154,Z 160.707,A -85,B 0,C 180,E1 -18145.886,E2 -18145.886} C_VEL
LIN {X 0,Y 263.128,Z 160.708,A -85,B 0,C 180,E1 -18149.504,E2 -18149.504} C_VEL
LIN {X 0,Y 263.144,Z 160.708,A -85,B 0,C 180,E1 -18152.997,E2 -18152.997} C_VEL
LIN {X 0,Y 263.146,Z 160.705,A -85,B 0,C 180,E1 -18156.383,E2 -18156.383} C_VEL
LIN {X 0,Y 263.21,Z 160.688,A -85,B 0,C 180,E1 -18159.689,E2 -18159.689} C_VEL
LIN {X 0,Y 263.291,Z 160.68,A -85,B 0,C 180,E1 -18164.518,E2 -18164.518} C_VEL
LIN {X 0,Y 263.33,Z 160.682,A -85,B 0,C 180,E1 -18169.233,E2 -18169.233} C_VEL
LIN {X 0,Y 263.516,Z 160.649,A -85,B 0,C 180,E1 -18172.337,E2 -18172.337} C_VEL
LIN {X 0,Y 263.727,Z 160.626,A -85,B 0,C 180,E1 -18178.473,E2 -18178.473} C_VEL
LIN {X 0,Y 263.733,Z 160.627,A -85,B 0,C 180,E1 -18181.527,E2 -18181.527} C_VEL
LIN {X 0,Y 263.528,Z 160.648,A -85,B 0,C 180,E1 -18187.663,E2 -18187.663} C_VEL
LIN {X 0,Y 263.352,Z 160.679,A -85,B 0,C 180,E1 -18190.767,E2 -18190.767} C_VEL
LIN {X 0,Y 263.313,Z 160.678,A -85,B 0,C 180,E1 -18195.481,E2 -18195.481} C_VEL
LIN {X 0,Y 263.212,Z 160.69,A -85,B 0,C 180,E1 -18200.311,E2 -18200.311} C_VEL
LIN {X 0,Y 263.173,Z 160.696,A -85,B 0,C 180,E1 -18205.295,E2 -18205.295} C_VEL
LIN {X 0,Y 263.14,Z 160.699,A -85,B 0,C 180,E1 -18208.735,E2 -18208.735} C_VEL
LIN {X 0,Y 263.132,Z 160.702,A -85,B 0,C 180,E1 -18212.289,E2 -18212.289} C_VEL
LIN {X 0,Y 263.187,Z 160.695,A -85,B 0,C 180,E1 -18216.763,E2 -18216.763} C_VEL
LIN {X 0,Y 263.128,Z 160.684,A -85,B 0,C 180,E1 -18221.593,E2 -18221.593} C_VEL
LIN {X 0,Y 263.127,Z 160.708,A -85,B 0,C 180,E1 -18226.016,E2 -18226.016} C_VEL
LIN {X 0,Y 263.109,Z 160.711,A -85,B 0,C 180,E1 -18230.127,E2 -18230.127} C_VEL
LIN {X 0,Y 263.194,Z 160.705,A -85,B 0,C 180,E1 -18231.478,E2 -18231.478} C_VEL
LIN {X 0,Y 264.145,Z 163.491,A -85,B 0,C 180,E1 -18231.72,E2 -18231.72} C_VEL
LIN {X 0,Y 265.74,Z 165.848,A -85,B 0,C 180,E1 -18232.045,E2 -18232.045} C_VEL
LIN {X 0,Y 271.349,Z 175.503,A -85,B 0,C 180,E1 -18233.189,E2 -18233.189} C_VEL
LIN {X 0,Y 279.577,Z 192.5,A -85,B 0,C 180,E1 -18234.844,E2 -18234.844} C_VEL
LIN {X 0,Y 283.655,Z 202.15,A -85,B 0,C 180,E1 -18235.654,E2 -18235.654} C_VEL
LIN {X 0,Y 281.345,Z 267.087,A -85,B 0,C 180,E1 -18237.302,E2 -18237.302} C_VEL
LIN {X 0,Y 280.371,Z 280.366,A -85,B 0,C 180,E1 -18237.919,E2 -18237.919} C_VEL
LIN {X 0,Y 278.857,Z 293.4,A -85,B 0,C 180,E1 -18238.815,E2 -18238.815} C_VEL
LIN {X 0,Y 277.192,Z 305.158,A -85,B 0,C 180,E1 -18239.95,E2 -18239.95} C_VEL
LIN {X 0,Y 275.141,Z 316.647,A -85,B 0,C 180,E1 -18241.383,E2 -18241.383} C_VEL
LIN {X 0,Y 272.821,Z 326.968,A -85,B 0,C 180,E1 -18242.996,E2 -18242.996} C_VEL
LIN {X 0,Y 270.997,Z 335.382,A -85,B 0,C 180,E1 -18244.664,E2 -18244.664} C_VEL
LIN {X 0,Y 269.05,Z 343.385,A -85,B 0,C 180,E1 -18246.605,E2 -18246.605} C_VEL
LIN {X 0,Y 267.039,Z 350.653,A -85,B 0,C 180,E1 -18248.783,E2 -18248.783} C_VEL
LIN {X 0,Y 265.064,Z 357.593,A -85,B 0,C 180,E1 -18251.446,E2 -18251.446} C_VEL
LIN {X 0,Y 263.822,Z 361.778,A -85,B 0,C 180,E1 -18253.54,E2 -18253.54} C_VEL
LIN {X 0,Y 262.732,Z 365.618,A -85,B 0,C 180,E1 -18256.068,E2 -18256.068} C_VEL
LIN {X 0,Y 262.162,Z 367.349,A -85,B 0,C 180,E1 -18257.615,E2 -18257.615} C_VEL
LIN {X 0,Y 261.537,Z 369.566,A -85,B 0,C 180,E1 -18260.72,E2 -18260.72} C_VEL
LIN {X 0,Y 261.418,Z 370.086,A -85,B 0,C 180,E1 -18262.274,E2 -18262.274} C_VEL
LIN {X 0,Y 261.424,Z 370.143,A -85,B 0,C 180,E1 -18264.097,E2 -18264.097} C_VEL
LIN {X 0,Y 261.321,Z 369.215,A -85,B 0,C 180,E1 -18266.915,E2 -18266.915} C_VEL
LIN {X 0,Y 261.305,Z 368.165,A -85,B 0,C 180,E1 -18268.457,E2 -18268.457} C_VEL
LIN {X 0,Y 261.435,Z 366.669,A -85,B 0,C 180,E1 -18269.999,E2 -18269.999} C_VEL
LIN {X 0,Y 261.955,Z 363.647,A -85,B 0,C 180,E1 -18272.305,E2 -18272.305} C_VEL
LIN {X 0,Y 262.533,Z 359.598,A -85,B 0,C 180,E1 -18274.605,E2 -18274.605} C_VEL
LIN {X 0,Y 263.467,Z 354.387,A -85,B 0,C 180,E1 -18276.893,E2 -18276.893} C_VEL
LIN {X 0,Y 264.528,Z 347.864,A -85,B 0,C 180,E1 -18279.171,E2 -18279.171} C_VEL
LIN {X 0,Y 265.864,Z 341.216,A -85,B 0,C 180,E1 -18281.048,E2 -18281.048} C_VEL
LIN {X 0,Y 267.29,Z 333.215,A -85,B 0,C 180,E1 -18282.913,E2 -18282.913} C_VEL
LIN {X 0,Y 269.056,Z 322.877,A -85,B 0,C 180,E1 -18284.858,E2 -18284.858} C_VEL
LIN {X 0,Y 270.595,Z 312.527,A -85,B 0,C 180,E1 -18286.405,E2 -18286.405} C_VEL
LIN {X 0,Y 272.269,Z 300.061,A -85,B 0,C 180,E1 -18287.848,E2 -18287.848} C_VEL
LIN {X 0,Y 273.442,Z 287.783,A -85,B 0,C 180,E1 -18288.933,E2 -18288.933} C_VEL
LIN {X 0,Y 274.415,Z 274.678,A -85,B 0,C 180,E1 -18289.738,E2 -18289.738} C_VEL
LIN {X 0,Y 274.981,Z 262.041,A -85,B 0,C 180,E1 -18290.231,E2 -18290.231} C_VEL
LIN {X 0,Y 276.859,Z 193.696,A -85,B 0,C 180,E1 -18291.976,E2 -18291.976} C_VEL
LIN {X 0,Y 270.873,Z 177.69,A -85,B 0,C 180,E1 -18293.033,E2 -18293.033} C_VEL
LIN {X 0,Y 265.757,Z 166.531,A -85,B 0,C 180,E1 -18293.907,E2 -18293.907} C_VEL
LIN {X 0,Y 263.296,Z 161.299,A -85,B 0,C 180,E1 -18294.338,E2 -18294.338} C_VEL
LIN {X 0,Y 263.209,Z 160.7,A -85,B 0,C 180,E1 -18294.395,E2 -18294.395} C_VEL
LIN {X 0,Y 263.178,Z 160.701,A -85,B 0,C 180,E1 -18298.728,E2 -18298.728} C_VEL
LIN {X 0,Y 263.131,Z 160.707,A -85,B 0,C 180,E1 -18302.286,E2 -18302.286} C_VEL
LIN {X 0,Y 263.183,Z 160.701,A -85,B 0,C 180,E1 -18305.976,E2 -18305.976} C_VEL
LIN {X 0,Y 263.102,Z 160.712,A -85,B 0,C 180,E1 -18309.871,E2 -18309.871} C_VEL
LIN {X 0,Y 263.118,Z 160.71,A -85,B 0,C 180,E1 -18313.982,E2 -18313.982} C_VEL
LIN {X 0,Y 263.119,Z 160.709,A -85,B 0,C 180,E1 -18318.405,E2 -18318.405} C_VEL
LIN {X 0,Y 263.178,Z 160.7,A -85,B 0,C 180,E1 -18323.235,E2 -18323.235} C_VEL
LIN {X 0,Y 263.126,Z 160.707,A -85,B 0,C 180,E1 -18327.71,E2 -18327.71} C_VEL
LIN {X 0,Y 263.171,Z 160.699,A -85,B 0,C 180,E1 -18331.791,E2 -18331.791} C_VEL
LIN {X 0,Y 263.19,Z 160.701,A -85,B 0,C 180,E1 -18335.212,E2 -18335.212} C_VEL
LIN {X 0,Y 263.226,Z 160.696,A -85,B 0,C 180,E1 -18339.69,E2 -18339.69} C_VEL
LIN {X 0,Y 263.301,Z 160.679,A -85,B 0,C 180,E1 -18344.519,E2 -18344.519} C_VEL
LIN {X 0,Y 263.336,Z 160.681,A -85,B 0,C 180,E1 -18349.233,E2 -18349.233} C_VEL
LIN {X 0,Y 263.515,Z 160.644,A -85,B 0,C 180,E1 -18352.337,E2 -18352.337} C_VEL
LIN {X 0,Y 263.467,Z 160.639,A -85,B 0,C 180,E1 -18353.774,E2 -18353.774} C_VEL
LIN {X 0,Y 262.852,Z 160.721,A -85,B 0,C 180,E1 -18355.051,E2 -18355.051} C_VEL
LIN {X 0,Y 260.11,Z 161.075,A -85,B 0,C 180,E1 -18357.137,E2 -18357.137} C_VEL
LIN {X 0,Y 257.761,Z 161.374,A -85,B 0,C 180,E1 -18358.832,E2 -18358.832} C_VEL
LIN {X 0,Y 256.748,Z 161.502,A -85,B 0,C 180,E1 -18360.145,E2 -18360.145} C_VEL
LIN {X 0,Y 256.663,Z 161.509,A -85,B 0,C 180,E1 -18360.589,E2 -18360.589} C_VEL
LIN {X 0,Y 256.44,Z 161.541,A -85,B 0,C 180,E1 -18363.142,E2 -18363.142} C_VEL
LIN {X 0,Y 256.458,Z 161.536,A -85,B 0,C 180,E1 -18367.875,E2 -18367.875} C_VEL
LIN {X 0,Y 256.277,Z 161.561,A -85,B 0,C 180,E1 -18371.067,E2 -18371.067} C_VEL
LIN {X 0,Y 256.221,Z 161.567,A -85,B 0,C 180,E1 -18375.92,E2 -18375.92} C_VEL
LIN {X 0,Y 256.139,Z 161.581,A -85,B 0,C 180,E1 -18380.897,E2 -18380.897} C_VEL
LIN {X 0,Y 256.159,Z 161.578,A -85,B 0,C 180,E1 -18385.129,E2 -18385.129} C_VEL
LIN {X 0,Y 256.091,Z 161.586,A -85,B 0,C 180,E1 -18389.602,E2 -18389.602} C_VEL
LIN {X 0,Y 256.06,Z 161.59,A -85,B 0,C 180,E1 -18393.294,E2 -18393.294} C_VEL
LIN {X 0,Y 256.107,Z 161.584,A -85,B 0,C 180,E1 -18397.272,E2 -18397.272} C_VEL
LIN {X 0,Y 256.048,Z 161.59,A -85,B 0,C 180,E1 -18401.205,E2 -18401.205} C_VEL
LIN {X 0,Y 256.052,Z 161.589,A -85,B 0,C 180,E1 -18405.532,E2 -18405.532} C_VEL
LIN {X 0,Y 256.049,Z 161.585,A -85,B 0,C 180,E1 -18408.798,E2 -18408.798} C_VEL
LIN {X 0,Y 256.19,Z 161.651,A -85,B 0,C 180,E1 -18413.555,E2 -18413.555} C_VEL
LIN {X 0,Y 258.556,Z 172.094,A -85,B 0,C 180,E1 -18417.419,E2 -18417.419} C_VEL
LIN {X 0,Y 260.26,Z 180.278,A -85,B 0,C 180,E1 -18420.284,E2 -18420.284} C_VEL
LIN {X 0,Y 263.959,Z 190.483,A -85,B 0,C 180,E1 -18421.001,E2 -18421.001} C_VEL
LIN {X 0,Y 267.652,Z 216.247,A -85,B 0,C 180,E1 -18422.147,E2 -18422.147} C_VEL
LIN {X 0,Y 269.425,Z 231.812,A -85,B 0,C 180,E1 -18422.774,E2 -18422.774} C_VEL
LIN {X 0,Y 267.709,Z 288.87,A -85,B 0,C 180,E1 -18424.281,E2 -18424.281} C_VEL
LIN {X 0,Y 266.854,Z 302.331,A -85,B 0,C 180,E1 -18424.924,E2 -18424.924} C_VEL
LIN {X 0,Y 265.511,Z 314.572,A -85,B 0,C 180,E1 -18425.779,E2 -18425.779} C_VEL
LIN {X 0,Y 263.989,Z 326.098,A -85,B 0,C 180,E1 -18426.881,E2 -18426.881} C_VEL
LIN {X 0,Y 262.187,Z 337.922,A -85,B 0,C 180,E1 -18428.374,E2 -18428.374} C_VEL
LIN {X 0,Y 260.228,Z 348.51,A -85,B 0,C 180,E1 -18430.066,E2 -18430.066} C_VEL
LIN {X 0,Y 258.616,Z 358.16,A -85,B 0,C 180,E1 -18432.016,E2 -18432.016} C_VEL
LIN {X 0,Y 257.123,Z 366.586,A -85,B 0,C 180,E1 -18434.139,E2 -18434.139} C_VEL
LIN {X 0,Y 255.839,Z 374.114,A -85,B 0,C 180,E1 -18436.499,E2 -18436.499} C_VEL
LIN {X 0,Y 254.898,Z 380.158,A -85,B 0,C 180,E1 -18438.874,E2 -18438.874} C_VEL
LIN {X 0,Y 254.354,Z 384.937,A -85,B 0,C 180,E1 -18441.261,E2 -18441.261} C_VEL
LIN {X 0,Y 254.148,Z 388.59,A -85,B 0,C 180,E1 -18443.651,E2 -18443.651} C_VEL
LIN {X 0,Y 254.067,Z 390.469,A -85,B 0,C 180,E1 -18445.241,E2 -18445.241} C_VEL
LIN {X 0,Y 254.11,Z 391.877,A -85,B 0,C 180,E1 -18446.831,E2 -18446.831} C_VEL
LIN {X 0,Y 254.137,Z 392.876,A -85,B 0,C 180,E1 -18448.417,E2 -18448.417} C_VEL
LIN {X 0,Y 254.168,Z 393.478,A -85,B 0,C 180,E1 -18450.001,E2 -18450.001} C_VEL
LIN {X 0,Y 254.119,Z 393.68,A -85,B 0,C 180,E1 -18451.586,E2 -18451.586} C_VEL
LIN {X 0,Y 254.054,Z 393.443,A -85,B 0,C 180,E1 -18453.173,E2 -18453.173} C_VEL
LIN {X 0,Y 254.057,Z 391.794,A -85,B 0,C 180,E1 -18456.354,E2 -18456.354} C_VEL
LIN {X 0,Y 254.249,Z 390.38,A -85,B 0,C 180,E1 -18457.946,E2 -18457.946} C_VEL
LIN {X 0,Y 254.767,Z 387.422,A -85,B 0,C 180,E1 -18460.331,E2 -18460.331} C_VEL
LIN {X 0,Y 255.623,Z 383.44,A -85,B 0,C 180,E1 -18462.707,E2 -18462.707} C_VEL
LIN {X 0,Y 257.332,Z 377.358,A -85,B 0,C 180,E1 -18465.444,E2 -18465.444} C_VEL
LIN {X 0,Y 259.373,Z 369.775,A -85,B 0,C 180,E1 -18468.06,E2 -18468.06} C_VEL
LIN {X 0,Y 261.163,Z 362.489,A -85,B 0,C 180,E1 -18470.068,E2 -18470.068} C_VEL
LIN {X 0,Y 263.389,Z 354.096,A -85,B 0,C 180,E1 -18471.937,E2 -18471.937} C_VEL
LIN {X 0,Y 265.911,Z 343.767,A -85,B 0,C 180,E1 -18473.77,E2 -18473.77} C_VEL
LIN {X 0,Y 268.5,Z 332.138,A -85,B 0,C 180,E1 -18475.381,E2 -18475.381} C_VEL
LIN {X 0,Y 270.662,Z 320.634,A -85,B 0,C 180,E1 -18476.611,E2 -18476.611} C_VEL
LIN {X 0,Y 272.669,Z 307.414,A -85,B 0,C 180,E1 -18477.643,E2 -18477.643} C_VEL
LIN {X 0,Y 274.153,Z 293.995,A -85,B 0,C 180,E1 -18478.364,E2 -18478.364} C_VEL
LIN {X 0,Y 274.877,Z 280.527,A -85,B 0,C 180,E1 -18478.804,E2 -18478.804} C_VEL
LIN {X 0,Y 276.41,Z 234.199,A -85,B 0,C 180,E1 -18479.995,E2 -18479.995} C_VEL
LIN {X 0,Y 272.755,Z 210.56,A -85,B 0,C 180,E1 -18481.198,E2 -18481.198} C_VEL
LIN {X 0,Y 271.122,Z 202.331,A -85,B 0,C 180,E1 -18481.679,E2 -18481.679} C_VEL
LIN {X 0,Y 264.146,Z 186.876,A -85,B 0,C 180,E1 -18483.191,E2 -18483.191} C_VEL
LIN {X 0,Y 260.652,Z 179.359,A -85,B 0,C 180,E1 -18484.019,E2 -18484.019} C_VEL
LIN {X 0,Y 258.31,Z 169.612,A -85,B 0,C 180,E1 -18487.906,E2 -18487.906} C_VEL
LIN {X 0,Y 256.094,Z 161.582,A -85,B 0,C 180,E1 -18491.403,E2 -18491.403} C_VEL
LIN {X 0,Y 256.04,Z 161.591,A -85,B 0,C 180,E1 -18495.536,E2 -18495.536} C_VEL
LIN {X 0,Y 256.042,Z 161.592,A -85,B 0,C 180,E1 -18498.794,E2 -18498.794} C_VEL
LIN {X 0,Y 256.128,Z 161.581,A -85,B 0,C 180,E1 -18502.867,E2 -18502.867} C_VEL
LIN {X 0,Y 256.069,Z 161.589,A -85,B 0,C 180,E1 -18506.707,E2 -18506.707} C_VEL
LIN {X 0,Y 256.057,Z 161.59,A -85,B 0,C 180,E1 -18510.393,E2 -18510.393} C_VEL
LIN {X 0,Y 256.135,Z 161.58,A -85,B 0,C 180,E1 -18514.889,E2 -18514.889} C_VEL
LIN {X 0,Y 256.126,Z 161.574,A -85,B 0,C 180,E1 -18519.101,E2 -18519.101} C_VEL
LIN {X 0,Y 256.216,Z 161.566,A -85,B 0,C 180,E1 -18524.08,E2 -18524.08} C_VEL
LIN {X 0,Y 256.274,Z 161.561,A -85,B 0,C 180,E1 -18528.933,E2 -18528.933} C_VEL
LIN {X 0,Y 256.458,Z 161.526,A -85,B 0,C 180,E1 -18532.125,E2 -18532.125} C_VEL
LIN {X 0,Y 256.292,Z 161.559,A -85,B 0,C 180,E1 -18535.281,E2 -18535.281} C_VEL
LIN {X 0,Y 256.688,Z 161.502,A -85,B 0,C 180,E1 -18538.431,E2 -18538.431} C_VEL
LIN {X 0,Y 256.695,Z 161.502,A -85,B 0,C 180,E1 -18541.569,E2 -18541.569} C_VEL
LIN {X 0,Y 256.444,Z 161.536,A -85,B 0,C 180,E1 -18546.572,E2 -18546.572} C_VEL
LIN {X 0,Y 256.43,Z 161.53,A -85,B 0,C 180,E1 -18549.465,E2 -18549.465} C_VEL
LIN {X 0,Y 256.234,Z 161.553,A -85,B 0,C 180,E1 -18554.292,E2 -18554.292} C_VEL
LIN {X 0,Y 256.166,Z 161.574,A -85,B 0,C 180,E1 -18557.565,E2 -18557.565} C_VEL
LIN {X 0,Y 256.126,Z 161.577,A -85,B 0,C 180,E1 -18561.099,E2 -18561.099} C_VEL
LIN {X 0,Y 256.137,Z 161.571,A -85,B 0,C 180,E1 -18565.112,E2 -18565.112} C_VEL
LIN {X 0,Y 256.06,Z 161.584,A -85,B 0,C 180,E1 -18569.607,E2 -18569.607} C_VEL
LIN {X 0,Y 256.07,Z 161.582,A -85,B 0,C 180,E1 -18573.293,E2 -18573.293} C_VEL
LIN {X 0,Y 256.119,Z 161.578,A -85,B 0,C 180,E1 -18577.271,E2 -18577.271} C_VEL
LIN {X 0,Y 256.058,Z 161.563,A -85,B 0,C 180,E1 -18581.203,E2 -18581.203} C_VEL
LIN {X 0,Y 256.062,Z 161.586,A -85,B 0,C 180,E1 -18585.53,E2 -18585.53} C_VEL
LIN {X 0,Y 256.058,Z 161.591,A -85,B 0,C 180,E1 -18588.796,E2 -18588.796} C_VEL
LIN {X 0,Y 256.088,Z 161.623,A -85,B 0,C 180,E1 -18590.341,E2 -18590.341} C_VEL
LIN {X 0,Y 257.027,Z 164.362,A -85,B 0,C 180,E1 -18590.594,E2 -18590.594} C_VEL
LIN {X 0,Y 258.669,Z 166.544,A -85,B 0,C 180,E1 -18590.942,E2 -18590.942} C_VEL
LIN {X 0,Y 266.397,Z 179.774,A -85,B 0,C 180,E1 -18592.596,E2 -18592.596} C_VEL
LIN {X 0,Y 274.253,Z 196.229,A -85,B 0,C 180,E1 -18594.242,E2 -18594.242} C_VEL
LIN {X 0,Y 277.586,Z 204.074,A -85,B 0,C 180,E1 -18594.929,E2 -18594.929} C_VEL
LIN {X 0,Y 275.208,Z 267.898,A -85,B 0,C 180,E1 -18596.588,E2 -18596.588} C_VEL
LIN {X 0,Y 274.078,Z 281.776,A -85,B 0,C 180,E1 -18597.254,E2 -18597.254} C_VEL
LIN {X 0,Y 272.518,Z 294.696,A -85,B 0,C 180,E1 -18598.194,E2 -18598.194} C_VEL
LIN {X 0,Y 270.742,Z 306.445,A -85,B 0,C 180,E1 -18599.373,E2 -18599.373} C_VEL
LIN {X 0,Y 268.607,Z 317.756,A -85,B 0,C 180,E1 -18600.835,E2 -18600.835} C_VEL
LIN {X 0,Y 266.209,Z 327.899,A -85,B 0,C 180,E1 -18602.482,E2 -18602.482} C_VEL
LIN {X 0,Y 264.102,Z 337.02,A -85,B 0,C 180,E1 -18604.377,E2 -18604.377} C_VEL
LIN {X 0,Y 261.867,Z 345.88,A -85,B 0,C 180,E1 -18606.679,E2 -18606.679} C_VEL
LIN {X 0,Y 259.725,Z 352.964,A -85,B 0,C 180,E1 -18608.988,E2 -18608.988} C_VEL
LIN {X 0,Y 257.76,Z 359.388,A -85,B 0,C 180,E1 -18611.725,E2 -18611.725} C_VEL
LIN {X 0,Y 256.434,Z 363.61,A -85,B 0,C 180,E1 -18614.092,E2 -18614.092} C_VEL
LIN {X 0,Y 255.787,Z 365.84,A -85,B 0,C 180,E1 -18615.682,E2 -18615.682} C_VEL
LIN {X 0,Y 255.172,Z 367.603,A -85,B 0,C 180,E1 -18617.27,E2 -18617.27} C_VEL
LIN {X 0,Y 254.487,Z 369.852,A -85,B 0,C 180,E1 -18620.461,E2 -18620.461} C_VEL
LIN {X 0,Y 254.341,Z 370.392,A -85,B 0,C 180,E1 -18622.057,E2 -18622.057} C_VEL
LIN {X 0,Y 254.342,Z 370.454,A -85,B 0,C 180,E1 -18624.134,E2 -18624.134} C_VEL
LIN {X 0,Y 254.229,Z 369.578,A -85,B 0,C 180,E1 -18626.829,E2 -18626.829} C_VEL
LIN {X 0,Y 254.228,Z 368.546,A -85,B 0,C 180,E1 -18628.414,E2 -18628.414} C_VEL
LIN {X 0,Y 254.347,Z 367.08,A -85,B 0,C 180,E1 -18629.999,E2 -18629.999} C_VEL
LIN {X 0,Y 254.867,Z 364.092,A -85,B 0,C 180,E1 -18632.369,E2 -18632.369} C_VEL
LIN {X 0,Y 255.473,Z 360.079,A -85,B 0,C 180,E1 -18634.732,E2 -18634.732} C_VEL
LIN {X 0,Y 256.448,Z 354.907,A -85,B 0,C 180,E1 -18637.082,E2 -18637.082} C_VEL
LIN {X 0,Y 257.547,Z 348.428,A -85,B 0,C 180,E1 -18639.422,E2 -18639.422} C_VEL
LIN {X 0,Y 259.258,Z 340.352,A -85,B 0,C 180,E1 -18641.729,E2 -18641.729} C_VEL
LIN {X 0,Y 260.756,Z 332.117,A -85,B 0,C 180,E1 -18643.639,E2 -18643.639} C_VEL
LIN {X 0,Y 262.522,Z 322.006,A -85,B 0,C 180,E1 -18645.526,E2 -18645.526} C_VEL
LIN {X 0,Y 264.27,Z 310.574,A -85,B 0,C 180,E1 -18647.207,E2 -18647.207} C_VEL
LIN {X 0,Y 265.772,Z 299.324,A -85,B 0,C 180,E1 -18648.499,E2 -18648.499} C_VEL
LIN {X 0,Y 266.909,Z 287.841,A -85,B 0,C 180,E1 -18649.515,E2 -18649.515} C_VEL
LIN {X 0,Y 267.886,Z 274.625,A -85,B 0,C 180,E1 -18650.34,E2 -18650.34} C_VEL
LIN {X 0,Y 268.504,Z 261.735,A -85,B 0,C 180,E1 -18650.841,E2 -18650.841} C_VEL
LIN {X 0,Y 270.48,Z 195.815,A -85,B 0,C 180,E1 -18652.549,E2 -18652.549} C_VEL
LIN {X 0,Y 265.869,Z 182.885,A -85,B 0,C 180,E1 -18653.41,E2 -18653.41} C_VEL
LIN {X 0,Y 260.463,Z 170.788,A -85,B 0,C 180,E1 -18654.372,E2 -18654.372} C_VEL
LIN {X 0,Y 256.317,Z 162.389,A -85,B 0,C 180,E1 -18655.117,E2 -18655.117} C_VEL
LIN {X 0,Y 256.159,Z 161.577,A -85,B 0,C 180,E1 -18655.225,E2 -18655.225} C_VEL
LIN {X 0,Y 256.112,Z 161.581,A -85,B 0,C 180,E1 -18659.598,E2 -18659.598} C_VEL
LIN {X 0,Y 256.083,Z 161.583,A -85,B 0,C 180,E1 -18663.288,E2 -18663.288} C_VEL
LIN {X 0,Y 256.123,Z 161.578,A -85,B 0,C 180,E1 -18667.272,E2 -18667.272} C_VEL
LIN {X 0,Y 256.067,Z 161.589,A -85,B 0,C 180,E1 -18672.179,E2 -18672.179} C_VEL
LIN {X 0,Y 256.056,Z 161.586,A -85,B 0,C 180,E1 -18676.671,E2 -18676.671} C_VEL
LIN {X 0,Y 256.066,Z 161.586,A -85,B 0,C 180,E1 -18680.856,E2 -18680.856} C_VEL
LIN {X 0,Y 256.126,Z 161.577,A -85,B 0,C 180,E1 -18682.866,E2 -18682.866} C_VEL
LIN {X 0,Y 256.061,Z 161.584,A -85,B 0,C 180,E1 -18686.706,E2 -18686.706} C_VEL
LIN {X 0,Y 256.092,Z 161.584,A -85,B 0,C 180,E1 -18690.397,E2 -18690.397} C_VEL
LIN {X 0,Y 256.159,Z 161.575,A -85,B 0,C 180,E1 -18694.871,E2 -18694.871} C_VEL
LIN {X 0,Y 256.139,Z 161.573,A -85,B 0,C 180,E1 -18699.102,E2 -18699.102} C_VEL
LIN {X 0,Y 256.221,Z 161.561,A -85,B 0,C 180,E1 -18704.08,E2 -18704.08} C_VEL
LIN {X 0,Y 256.278,Z 161.562,A -85,B 0,C 180,E1 -18708.932,E2 -18708.932} C_VEL
LIN {X 0,Y 256.457,Z 161.522,A -85,B 0,C 180,E1 -18712.124,E2 -18712.124} C_VEL
LIN {X 0,Y 256.437,Z 161.53,A -85,B 0,C 180,E1 -18716.858,E2 -18716.858} C_VEL
LIN {X 0,Y 256.684,Z 161.506,A -85,B 0,C 180,E1 -18718.431,E2 -18718.431} C_VEL
LIN {X 0,Y 256.663,Z 161.509,A -85,B 0,C 180,E1 -18720.589,E2 -18720.589} C_VEL
LIN {X 0,Y 255.963,Z 161.599,A -85,B 0,C 180,E1 -18721.895,E2 -18721.895} C_VEL
LIN {X 0,Y 253.011,Z 161.967,A -85,B 0,C 180,E1 -18724.021,E2 -18724.021} C_VEL
LIN {X 0,Y 250.519,Z 162.278,A -85,B 0,C 180,E1 -18725.752,E2 -18725.752} C_VEL
LIN {X 0,Y 249.464,Z 162.409,A -85,B 0,C 180,E1 -18727.097,E2 -18727.097} C_VEL
LIN {X 0,Y 249.386,Z 162.415,A -85,B 0,C 180,E1 -18727.553,E2 -18727.553} C_VEL
LIN {X 0,Y 249.324,Z 162.428,A -85,B 0,C 180,E1 -18729.737,E2 -18729.737} C_VEL
LIN {X 0,Y 249.162,Z 162.452,A -85,B 0,C 180,E1 -18734.706,E2 -18734.706} C_VEL
LIN {X 0,Y 249.094,Z 162.458,A -85,B 0,C 180,E1 -18738.081,E2 -18738.081} C_VEL
LIN {X 0,Y 249.071,Z 162.46,A -85,B 0,C 180,E1 -18741.519,E2 -18741.519} C_VEL
LIN {X 0,Y 249.105,Z 162.456,A -85,B 0,C 180,E1 -18745.475,E2 -18745.475} C_VEL
LIN {X 0,Y 249.056,Z 162.463,A -85,B 0,C 180,E1 -18748.986,E2 -18748.986} C_VEL
LIN {X 0,Y 249.023,Z 162.471,A -85,B 0,C 180,E1 -18752.427,E2 -18752.427} C_VEL
LIN {X 0,Y 249.041,Z 162.467,A -85,B 0,C 180,E1 -18756.344,E2 -18756.344} C_VEL
LIN {X 0,Y 248.999,Z 162.471,A -85,B 0,C 180,E1 -18760.479,E2 -18760.479} C_VEL
LIN {X 0,Y 248.996,Z 162.468,A -85,B 0,C 180,E1 -18764.881,E2 -18764.881} C_VEL
LIN {X 0,Y 249.01,Z 162.461,A -85,B 0,C 180,E1 -18767.364,E2 -18767.364} C_VEL
LIN {X 0,Y 249.046,Z 162.464,A -85,B 0,C 180,E1 -18772.2,E2 -18772.2} C_VEL
LIN {X 0,Y 249.111,Z 162.584,A -85,B 0,C 180,E1 -18772.915,E2 -18772.915} C_VEL
LIN {X 0,Y 251.56,Z 173.072,A -85,B 0,C 180,E1 -18776.943,E2 -18776.943} C_VEL
LIN {X 0,Y 253.026,Z 180.134,A -85,B 0,C 180,E1 -18779.435,E2 -18779.435} C_VEL
LIN {X 0,Y 257.798,Z 192.756,A -85,B 0,C 180,E1 -18780.386,E2 -18780.386} C_VEL
LIN {X 0,Y 261.389,Z 218.324,A -85,B 0,C 180,E1 -18781.557,E2 -18781.557} C_VEL
LIN {X 0,Y 262.96,Z 233.578,A -85,B 0,C 180,E1 -18782.175,E2 -18782.175} C_VEL
LIN {X 0,Y 261.176,Z 289.458,A -85,B 0,C 180,E1 -18783.696,E2 -18783.696} C_VEL
LIN {X 0,Y 260.203,Z 303.372,A -85,B 0,C 180,E1 -18784.398,E2 -18784.398} C_VEL
LIN {X 0,Y 258.757,Z 315.795,A -85,B 0,C 180,E1 -18785.319,E2 -18785.319} C_VEL
LIN {X 0,Y 256.933,Z 328.494,A -85,B 0,C 180,E1 -18786.635,E2 -18786.635} C_VEL
LIN {X 0,Y 255.101,Z 339.803,A -85,B 0,C 180,E1 -18788.168,E2 -18788.168} C_VEL
LIN {X 0,Y 253.191,Z 349.967,A -85,B 0,C 180,E1 -18789.911,E2 -18789.911} C_VEL
LIN {X 0,Y 251.412,Z 359.979,A -85,B 0,C 180,E1 -18792.094,E2 -18792.094} C_VEL
LIN {X 0,Y 249.98,Z 367.421,A -85,B 0,C 180,E1 -18794.093,E2 -18794.093} C_VEL
LIN {X 0,Y 248.681,Z 374.745,A -85,B 0,C 180,E1 -18796.519,E2 -18796.519} C_VEL
LIN {X 0,Y 247.887,Z 379.694,A -85,B 0,C 180,E1 -18798.555,E2 -18798.555} C_VEL
LIN {X 0,Y 247.308,Z 384.503,A -85,B 0,C 180,E1 -18801.009,E2 -18801.009} C_VEL
LIN {X 0,Y 247.053,Z 388.183,A -85,B 0,C 180,E1 -18803.468,E2 -18803.468} C_VEL
LIN {X 0,Y 246.99,Z 390.081,A -85,B 0,C 180,E1 -18805.105,E2 -18805.105} C_VEL
LIN {X 0,Y 247.022,Z 391.511,A -85,B 0,C 180,E1 -18806.74,E2 -18806.74} C_VEL
LIN {X 0,Y 247.064,Z 392.522,A -85,B 0,C 180,E1 -18808.371,E2 -18808.371} C_VEL
LIN {X 0,Y 247.092,Z 393.137,A -85,B 0,C 180,E1 -18810.001,E2 -18810.001} C_VEL
LIN {X 0,Y 247.045,Z 393.355,A -85,B 0,C 180,E1 -18811.632,E2 -18811.632} C_VEL
LIN {X 0,Y 246.967,Z 393.137,A -85,B 0,C 180,E1 -18813.264,E2 -18813.264} C_VEL
LIN {X 0,Y 246.977,Z 391.511,A -85,B 0,C 180,E1 -18816.537,E2 -18816.537} C_VEL
LIN {X 0,Y 247.187,Z 390.113,A -85,B 0,C 180,E1 -18818.174,E2 -18818.174} C_VEL
LIN {X 0,Y 247.761,Z 387.178,A -85,B 0,C 180,E1 -18820.626,E2 -18820.626} C_VEL
LIN {X 0,Y 248.661,Z 383.223,A -85,B 0,C 180,E1 -18823.069,E2 -18823.069} C_VEL
LIN {X 0,Y 250.174,Z 378.157,A -85,B 0,C 180,E1 -18825.48,E2 -18825.48} C_VEL
LIN {X 0,Y 252.001,Z 371.809,A -85,B 0,C 180,E1 -18827.866,E2 -18827.866} C_VEL
LIN {X 0,Y 254.071,Z 363.879,A -85,B 0,C 180,E1 -18830.23,E2 -18830.23} C_VEL
LIN {X 0,Y 256.307,Z 355.826,A -85,B 0,C 180,E1 -18832.151,E2 -18832.151} C_VEL
LIN {X 0,Y 258.913,Z 346.021,A -85,B 0,C 180,E1 -18834.028,E2 -18834.028} C_VEL
LIN {X 0,Y 261.51,Z 335.097,A -85,B 0,C 180,E1 -18835.682,E2 -18835.682} C_VEL
LIN {X 0,Y 263.664,Z 324.407,A -85,B 0,C 180,E1 -18836.946,E2 -18836.946} C_VEL
LIN {X 0,Y 265.915,Z 311.542,A -85,B 0,C 180,E1 -18838.086,E2 -18838.086} C_VEL
LIN {X 0,Y 267.605,Z 298.46,A -85,B 0,C 180,E1 -18838.909,E2 -18838.909} C_VEL
LIN {X 0,Y 268.572,Z 285.423,A -85,B 0,C 180,E1 -18839.438,E2 -18839.438} C_VEL
